KUKA KRL program: EPS_2_251292_SANCTRLMH1A_A_20251205052954.src

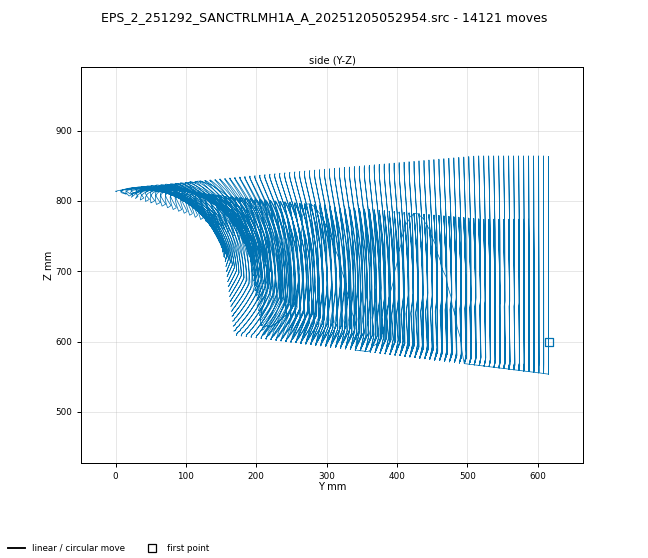
[picture p0: tool path of EPS_2_251292_SANCTRLMH1A_A_20251205052954.src, 14121 of 14123 moves have a stored position in this frame; points joined in program order, loops and branches not executed]
&ACCESS RVP
&REL 4
&COMMENT QRS 19112012
&PARAM EDITMASK = *
DEF PART()
EXT BAS (BAS_COMMAND :IN,REAL :IN )
INT I
BAS (#INITMOV,0 )

;KUKA QRS Post kuka4.cps  Date:22-06-2017 !

File_ID=2942

QRS_PRE_INIT()

;Init var - Until changes are made in qrs_pre_init
Outlet_Square_prg=0
Inlet_1_Square_prg=0
Inlet_2_Square_prg=0
Inlet_3_Square_prg=0
Inlet_4_Square_prg=0
Inlet_5_Square_prg=0

Outlet_1={X 0.000, Y 513.730, Z 763.500, B 0.000, E1 0.000 }
Inlet_1={X 0.000, Y 520.160, Z 673.500, B 0.000, E1 168.000 }
Inlet_2={X 0.000, Y 520.160, Z 673.500, B 0.000, E1 226.000 }
Outlet_1_type=201
Inlet_1_type=201
Inlet_2_type=201
;QRS#1=Sidecore dimensions
;QRS#2=200-8" PVC SDR 35
;QRS#3=200-8" PVC SDR 35
;QRS#4=200-8" PVC SDR 35
;QRS#5=
;QRS#6=
;QRS#7=
;QRS#8=
;QRS#9=12-08 PSX
;QRS#10=12-08 PSX
;QRS#11=12-08 PSX
;QRS#12=
;QRS#13=
;QRS#14=
;QRS#15=
;QRS#16=1220x127x1143 3,75'
;QRS#17=EPS Height
;QRS#18=864
;QRS#19=*
;QRS#20= UPDATED VERSION 22-06-2017
;QRS#21=*
Outlet_Square=0100
Inlet_1_Square=0100
Inlet_2_Square=0100
Inlet_3_Square=0
Inlet_4_Square=0
Inlet_5_Square=0
Mill_Square=1
Outlet_Square_Prg=204
Inlet_1_Square_prg=204
Inlet_2_Square_prg=204

QRS_INIT()

$ADVANCE=5

; T1
PTP {E1 173.592,E2 173.592}
PTP {X 0,Y 615.51,A -85,B 0,C 180,E1 173.592,E2 173.592,E3 0,E4 0,E5 0,E6 0}
QRS_SPEED_INIT()
LIN {X 0,Y 615.51,Z 600,A -85,B 0,C 180,E1 173.592,E2 173.592,E3 0,E4 0,E5 0,E6 0} C_VEL
LIN {X 0,Y 615.51,Z 563.866,A -85,B 0,C 180,E1 173.592,E2 173.592} C_VEL
LIN {X 0,Y 615.51,Z 555.694,A -85,B 0,C 180,E1 173.592,E2 173.592} C_VEL
LIN {X 0,Y 615.492,Z 553.694,A -85,B 0,C 180,E1 173.406,E2 173.406} C_VEL
LIN {X 0,Y 615.478,Z 553.692,A -85,B 0,C 180,E1 170.801,E2 170.801} C_VEL
LIN {X 0,Y 615.485,Z 553.682,A -85,B 0,C 180,E1 168.139,E2 168.139} C_VEL
LIN {X 0,Y 615.482,Z 553.692,A -85,B 0,C 180,E1 165.451,E2 165.451} C_VEL
LIN {X 0,Y 615.481,Z 553.693,A -85,B 0,C 180,E1 162.729,E2 162.729} C_VEL
LIN {X 0,Y 615.485,Z 553.682,A -85,B 0,C 180,E1 159.967,E2 159.967} C_VEL
LIN {X 0,Y 615.487,Z 553.696,A -85,B 0,C 180,E1 157.155,E2 157.155} C_VEL
LIN {X 0,Y 615.484,Z 553.684,A -85,B 0,C 180,E1 154.284,E2 154.284} C_VEL
LIN {X 0,Y 615.476,Z 553.687,A -85,B 0,C 180,E1 151.549,E2 151.549} C_VEL
LIN {X 0,Y 615.483,Z 553.703,A -85,B 0,C 180,E1 148.912,E2 148.912} C_VEL
LIN {X 0,Y 615.496,Z 553.68,A -85,B 0,C 180,E1 145.978,E2 145.978} C_VEL
LIN {X 0,Y 615.482,Z 553.694,A -85,B 0,C 180,E1 143.062,E2 143.062} C_VEL
LIN {X 0,Y 615.477,Z 553.689,A -85,B 0,C 180,E1 140.249,E2 140.249} C_VEL
LIN {X 0,Y 615.488,Z 553.681,A -85,B 0,C 180,E1 137.647,E2 137.647} C_VEL
LIN {X 0,Y 615.479,Z 553.696,A -85,B 0,C 180,E1 134.93,E2 134.93} C_VEL
LIN {X 0,Y 615.477,Z 553.687,A -85,B 0,C 180,E1 132.079,E2 132.079} C_VEL
LIN {X 0,Y 615.493,Z 553.68,A -85,B 0,C 180,E1 129.749,E2 129.749} C_VEL
LIN {X 0,Y 615.477,Z 553.693,A -85,B 0,C 180,E1 126.935,E2 126.935} C_VEL
LIN {X 0,Y 615.489,Z 553.697,A -85,B 0,C 180,E1 124.7,E2 124.7} C_VEL
LIN {X 0,Y 615.484,Z 553.696,A -85,B 0,C 180,E1 122.33,E2 122.33} C_VEL
LIN {X 0,Y 615.493,Z 553.68,A -85,B 0,C 180,E1 119.405,E2 119.405} C_VEL
LIN {X 0,Y 615.477,Z 553.849,A -85,B 0,C 180,E1 116.93,E2 116.93} C_VEL
LIN {X 0,Y 615.484,Z 564.333,A -85,B 0,C 180,E1 114.811,E2 114.811} C_VEL
LIN {X 0,Y 615.489,Z 670.429,A -85,B 0,C 180,E1 113.533,E2 113.533} C_VEL
LIN {X 0,Y 615.487,Z 683.41,A -85,B 0,C 180,E1 113.244,E2 113.244} C_VEL
LIN {X 0,Y 615.487,Z 695.565,A -85,B 0,C 180,E1 112.844,E2 112.844} C_VEL
LIN {X 0,Y 615.488,Z 707.887,A -85,B 0,C 180,E1 112.294,E2 112.294} C_VEL
LIN {X 0,Y 615.482,Z 719.67,A -85,B 0,C 180,E1 111.607,E2 111.607} C_VEL
LIN {X 0,Y 615.499,Z 730.452,A -85,B 0,C 180,E1 110.817,E2 110.817} C_VEL
LIN {X 0,Y 615.497,Z 739.119,A -85,B 0,C 180,E1 110.032,E2 110.032} C_VEL
LIN {X 0,Y 615.496,Z 748.438,A -85,B 0,C 180,E1 108.991,E2 108.991} C_VEL
LIN {X 0,Y 615.498,Z 755.797,A -85,B 0,C 180,E1 107.956,E2 107.956} C_VEL
LIN {X 0,Y 615.496,Z 761.581,A -85,B 0,C 180,E1 106.928,E2 106.928} C_VEL
LIN {X 0,Y 615.496,Z 766.062,A -85,B 0,C 180,E1 105.905,E2 105.905} C_VEL
LIN {X 0,Y 615.495,Z 768.406,A -85,B 0,C 180,E1 105.225,E2 105.225} C_VEL
LIN {X 0,Y 615.497,Z 770.293,A -85,B 0,C 180,E1 104.548,E2 104.548} C_VEL
LIN {X 0,Y 615.495,Z 771.682,A -85,B 0,C 180,E1 103.874,E2 103.874} C_VEL
LIN {X 0,Y 615.499,Z 772.654,A -85,B 0,C 180,E1 103.201,E2 103.201} C_VEL
LIN {X 0,Y 615.495,Z 773.23,A -85,B 0,C 180,E1 102.53,E2 102.53} C_VEL
LIN {X 0,Y 615.496,Z 773.372,A -85,B 0,C 180,E1 101.86,E2 101.86} C_VEL
LIN {X 0,Y 615.495,Z 772.439,A -85,B 0,C 180,E1 100.527,E2 100.527} C_VEL
LIN {X 0,Y 615.499,Z 771.379,A -85,B 0,C 180,E1 99.862,E2 99.862} C_VEL
LIN {X 0,Y 615.495,Z 769.863,A -85,B 0,C 180,E1 99.198,E2 99.198} C_VEL
LIN {X 0,Y 615.495,Z 766.811,A -85,B 0,C 180,E1 98.206,E2 98.206} C_VEL
LIN {X 0,Y 615.496,Z 762.717,A -85,B 0,C 180,E1 97.215,E2 97.215} C_VEL
LIN {X 0,Y 615.496,Z 756.461,A -85,B 0,C 180,E1 96.063,E2 96.063} C_VEL
LIN {X 0,Y 615.496,Z 749.669,A -85,B 0,C 180,E1 95.077,E2 95.077} C_VEL
LIN {X 0,Y 615.499,Z 741.216,A -85,B 0,C 180,E1 94.092,E2 94.092} C_VEL
LIN {X 0,Y 615.497,Z 732.559,A -85,B 0,C 180,E1 93.273,E2 93.273} C_VEL
LIN {X 0,Y 615.496,Z 721.959,A -85,B 0,C 180,E1 92.454,E2 92.454} C_VEL
LIN {X 0,Y 615.487,Z 711.331,A -85,B 0,C 180,E1 91.799,E2 91.799} C_VEL
LIN {X 0,Y 615.492,Z 699.51,A -85,B 0,C 180,E1 91.227,E2 91.227} C_VEL
LIN {X 0,Y 615.478,Z 687.237,A -85,B 0,C 180,E1 90.777,E2 90.777} C_VEL
LIN {X 0,Y 615.474,Z 674.443,A -85,B 0,C 180,E1 90.45,E2 90.45} C_VEL
LIN {X 0,Y 615.483,Z 659.053,A -85,B 0,C 180,E1 90.225,E2 90.225} C_VEL
LIN {X 0,Y 615.487,Z 563.524,A -85,B 0,C 180,E1 89.1,E2 89.1} C_VEL
LIN {X 0,Y 615.477,Z 553.688,A -85,B 0,C 180,E1 87.341,E2 87.341} C_VEL
LIN {X 0,Y 615.485,Z 553.683,A -85,B 0,C 180,E1 84.759,E2 84.759} C_VEL
LIN {X 0,Y 615.484,Z 553.697,A -85,B 0,C 180,E1 82.125,E2 82.125} C_VEL
LIN {X 0,Y 615.477,Z 553.69,A -85,B 0,C 180,E1 79.473,E2 79.473} C_VEL
LIN {X 0,Y 615.497,Z 553.68,A -85,B 0,C 180,E1 76.799,E2 76.799} C_VEL
LIN {X 0,Y 615.487,Z 553.698,A -85,B 0,C 180,E1 74.095,E2 74.095} C_VEL
LIN {X 0,Y 615.477,Z 553.688,A -85,B 0,C 180,E1 71.354,E2 71.354} C_VEL
LIN {X 0,Y 615.492,Z 553.684,A -85,B 0,C 180,E1 68.569,E2 68.569} C_VEL
LIN {X 0,Y 615.497,Z 553.692,A -85,B 0,C 180,E1 65.729,E2 65.729} C_VEL
LIN {X 0,Y 615.479,Z 553.684,A -85,B 0,C 180,E1 62.823,E2 62.823} C_VEL
LIN {X 0,Y 615.48,Z 553.696,A -85,B 0,C 180,E1 60.207,E2 60.207} C_VEL
LIN {X 0,Y 615.488,Z 553.688,A -85,B 0,C 180,E1 58.542,E2 58.542} C_VEL
LIN {X 0,Y 615.478,Z 563.8,A -85,B 0,C 180,E1 56.801,E2 56.801} C_VEL
LIN {X 0,Y 615.49,Z 670.43,A -85,B 0,C 180,E1 55.533,E2 55.533} C_VEL
LIN {X 0,Y 615.491,Z 683.455,A -85,B 0,C 180,E1 55.243,E2 55.243} C_VEL
LIN {X 0,Y 615.489,Z 695.76,A -85,B 0,C 180,E1 54.837,E2 54.837} C_VEL
LIN {X 0,Y 615.493,Z 707.167,A -85,B 0,C 180,E1 54.331,E2 54.331} C_VEL
LIN {X 0,Y 615.478,Z 719.02,A -85,B 0,C 180,E1 53.65,E2 53.65} C_VEL
LIN {X 0,Y 615.498,Z 729.264,A -85,B 0,C 180,E1 52.911,E2 52.911} C_VEL
LIN {X 0,Y 615.495,Z 737.595,A -85,B 0,C 180,E1 52.181,E2 52.181} C_VEL
LIN {X 0,Y 615.496,Z 745.845,A -85,B 0,C 180,E1 51.307,E2 51.307} C_VEL
LIN {X 0,Y 615.494,Z 753.849,A -85,B 0,C 180,E1 50.252,E2 50.252} C_VEL
LIN {X 0,Y 615.495,Z 760.453,A -85,B 0,C 180,E1 49.151,E2 49.151} C_VEL
LIN {X 0,Y 615.495,Z 764.795,A -85,B 0,C 180,E1 48.224,E2 48.224} C_VEL
LIN {X 0,Y 615.495,Z 768.162,A -85,B 0,C 180,E1 47.302,E2 47.302} C_VEL
LIN {X 0,Y 615.493,Z 771.468,A -85,B 0,C 180,E1 46.002,E2 46.002} C_VEL
LIN {X 0,Y 615.493,Z 772.946,A -85,B 0,C 180,E1 44.933,E2 44.933} C_VEL
LIN {X 0,Y 615.492,Z 773.385,A -85,B 0,C 180,E1 43.999,E2 43.999} C_VEL
LIN {X 0,Y 615.494,Z 772.997,A -85,B 0,C 180,E1 43.05,E2 43.05} C_VEL
LIN {X 0,Y 615.494,Z 771.759,A -85,B 0,C 180,E1 42.082,E2 42.082} C_VEL
LIN {X 0,Y 615.495,Z 769.591,A -85,B 0,C 180,E1 41.097,E2 41.097} C_VEL
LIN {X 0,Y 615.496,Z 766.384,A -85,B 0,C 180,E1 40.092,E2 40.092} C_VEL
LIN {X 0,Y 615.494,Z 761.199,A -85,B 0,C 180,E1 38.904,E2 38.904} C_VEL
LIN {X 0,Y 615.497,Z 754.943,A -85,B 0,C 180,E1 37.82,E2 37.82} C_VEL
LIN {X 0,Y 615.493,Z 747.546,A -85,B 0,C 180,E1 36.81,E2 36.81} C_VEL
LIN {X 0,Y 615.498,Z 738.717,A -85,B 0,C 180,E1 35.837,E2 35.837} C_VEL
LIN {X 0,Y 615.497,Z 729.459,A -85,B 0,C 180,E1 35.014,E2 35.014} C_VEL
LIN {X 0,Y 615.49,Z 719.279,A -85,B 0,C 180,E1 34.277,E2 34.277} C_VEL
LIN {X 0,Y 615.48,Z 707.513,A -85,B 0,C 180,E1 33.596,E2 33.596} C_VEL
LIN {X 0,Y 615.49,Z 696.199,A -85,B 0,C 180,E1 33.09,E2 33.09} C_VEL
LIN {X 0,Y 615.478,Z 684.677,A -85,B 0,C 180,E1 32.701,E2 32.701} C_VEL
LIN {X 0,Y 615.478,Z 671.437,A -85,B 0,C 180,E1 32.395,E2 32.395} C_VEL
LIN {X 0,Y 615.489,Z 640.455,A -85,B 0,C 180,E1 32.008,E2 32.008} C_VEL
LIN {X 0,Y 615.486,Z 564.37,A -85,B 0,C 180,E1 31.107,E2 31.107} C_VEL
LIN {X 0,Y 615.49,Z 553.686,A -85,B 0,C 180,E1 28.938,E2 28.938} C_VEL
LIN {X 0,Y 615.476,Z 553.684,A -85,B 0,C 180,E1 26.445,E2 26.445} C_VEL
LIN {X 0,Y 615.485,Z 553.686,A -85,B 0,C 180,E1 24.011,E2 24.011} C_VEL
LIN {X 0,Y 615.499,Z 553.699,A -85,B 0,C 180,E1 21.432,E2 21.432} C_VEL
LIN {X 0,Y 615.483,Z 553.683,A -85,B 0,C 180,E1 18.608,E2 18.608} C_VEL
LIN {X 0,Y 615.483,Z 553.689,A -85,B 0,C 180,E1 15.905,E2 15.905} C_VEL
LIN {X 0,Y 615.488,Z 553.693,A -85,B 0,C 180,E1 13.201,E2 13.201} C_VEL
LIN {X 0,Y 615.485,Z 553.682,A -85,B 0,C 180,E1 10.527,E2 10.527} C_VEL
LIN {X 0,Y 615.482,Z 553.69,A -85,B 0,C 180,E1 7.876,E2 7.876} C_VEL
LIN {X 0,Y 615.486,Z 553.695,A -85,B 0,C 180,E1 5.241,E2 5.241} C_VEL
LIN {X 0,Y 615.494,Z 553.681,A -85,B 0,C 180,E1 2.618,E2 2.618} C_VEL
LIN {X 0,Y 615.476,Z 553.689,A -85,B 0,C 180,E1 0,E2 0} C_VEL
LIN {X 0,Y 615.494,Z 553.698,A -85,B 0,C 180,E1 -2.618,E2 -2.618} C_VEL
LIN {X 0,Y 615.478,Z 553.686,A -85,B 0,C 180,E1 -5.241,E2 -5.241} C_VEL
LIN {X 0,Y 615.485,Z 553.685,A -85,B 0,C 180,E1 -7.876,E2 -7.876} C_VEL
LIN {X 0,Y 615.493,Z 553.701,A -85,B 0,C 180,E1 -10.527,E2 -10.527} C_VEL
LIN {X 0,Y 615.476,Z 553.687,A -85,B 0,C 180,E1 -13.202,E2 -13.202} C_VEL
LIN {X 0,Y 615.487,Z 553.685,A -85,B 0,C 180,E1 -15.905,E2 -15.905} C_VEL
LIN {X 0,Y 615.493,Z 553.696,A -85,B 0,C 180,E1 -18.646,E2 -18.646} C_VEL
LIN {X 0,Y 615.476,Z 553.684,A -85,B 0,C 180,E1 -21.432,E2 -21.432} C_VEL
LIN {X 0,Y 615.492,Z 553.693,A -85,B 0,C 180,E1 -24.272,E2 -24.272} C_VEL
LIN {X 0,Y 615.48,Z 553.686,A -85,B 0,C 180,E1 -27.178,E2 -27.178} C_VEL
LIN {X 0,Y 615.485,Z 553.684,A -85,B 0,C 180,E1 -29.797,E2 -29.797} C_VEL
LIN {X 0,Y 615.494,Z 553.7,A -85,B 0,C 180,E1 -32.457,E2 -32.457} C_VEL
LIN {X 0,Y 615.485,Z 553.692,A -85,B 0,C 180,E1 -34.815,E2 -34.815} C_VEL
LIN {X 0,Y 615.49,Z 553.683,A -85,B 0,C 180,E1 -37.242,E2 -37.242} C_VEL
LIN {X 0,Y 615.493,Z 553.688,A -85,B 0,C 180,E1 -40.091,E2 -40.091} C_VEL
LIN {X 0,Y 615.485,Z 553.687,A -85,B 0,C 180,E1 -43.049,E2 -43.049} C_VEL
LIN {X 0,Y 615.477,Z 553.687,A -85,B 0,C 180,E1 -45.851,E2 -45.851} C_VEL
LIN {X 0,Y 615.49,Z 553.701,A -85,B 0,C 180,E1 -48.528,E2 -48.528} C_VEL
LIN {X 0,Y 615.482,Z 553.686,A -85,B 0,C 180,E1 -51.096,E2 -51.096} C_VEL
LIN {X 0,Y 615.481,Z 553.683,A -85,B 0,C 180,E1 -53.576,E2 -53.576} C_VEL
LIN {X 0,Y 615.498,Z 553.7,A -85,B 0,C 180,E1 -56.465,E2 -56.465} C_VEL
LIN {X 0,Y 615.477,Z 553.688,A -85,B 0,C 180,E1 -59.081,E2 -59.081} C_VEL
LIN {X 0,Y 615.494,Z 553.68,A -85,B 0,C 180,E1 -61.549,E2 -61.549} C_VEL
LIN {X 0,Y 615.494,Z 553.7,A -85,B 0,C 180,E1 -64.43,E2 -64.43} C_VEL
LIN {X 0,Y 615.491,Z 553.765,A -85,B 0,C 180,E1 -65.706,E2 -65.706} C_VEL
LIN {X 0,Y 615.495,Z 577.471,A -85,B 0,C 180,E1 -68.569,E2 -68.569} C_VEL
LIN {X 0,Y 615.483,Z 601.351,A -85,B 0,C 180,E1 -71.397,E2 -71.397} C_VEL
LIN {X 0,Y 615.478,Z 624.467,A -85,B 0,C 180,E1 -74.095,E2 -74.095} C_VEL
LIN {X 0,Y 615.486,Z 649.386,A -85,B 0,C 180,E1 -76.967,E2 -76.967} C_VEL
LIN {X 0,Y 615.48,Z 650.668,A -85,B 0,C 180,E1 -77.114,E2 -77.114} C_VEL
LIN {X 0,Y 615.476,Z 759.849,A -85,B 0,C 180,E1 -78.411,E2 -78.411} C_VEL
LIN {X 0,Y 615.487,Z 772.354,A -85,B 0,C 180,E1 -78.682,E2 -78.682} C_VEL
LIN {X 0,Y 615.496,Z 785.511,A -85,B 0,C 180,E1 -79.109,E2 -79.109} C_VEL
LIN {X 0,Y 615.484,Z 797.482,A -85,B 0,C 180,E1 -79.64,E2 -79.64} C_VEL
LIN {X 0,Y 615.483,Z 809,A -85,B 0,C 180,E1 -80.304,E2 -80.304} C_VEL
LIN {X 0,Y 615.499,Z 819.344,A -85,B 0,C 180,E1 -81.05,E2 -81.05} C_VEL
LIN {X 0,Y 615.497,Z 827.814,A -85,B 0,C 180,E1 -81.794,E2 -81.794} C_VEL
LIN {X 0,Y 615.498,Z 835.608,A -85,B 0,C 180,E1 -82.62,E2 -82.62} C_VEL
LIN {X 0,Y 615.496,Z 843.204,A -85,B 0,C 180,E1 -83.608,E2 -83.608} C_VEL
LIN {X 0,Y 615.498,Z 850.205,A -85,B 0,C 180,E1 -84.759,E2 -84.759} C_VEL
LIN {X 0,Y 615.494,Z 854.852,A -85,B 0,C 180,E1 -85.744,E2 -85.744} C_VEL
LIN {X 0,Y 615.496,Z 858.399,A -85,B 0,C 180,E1 -86.727,E2 -86.727} C_VEL
LIN {X 0,Y 615.497,Z 860.233,A -85,B 0,C 180,E1 -87.382,E2 -87.382} C_VEL
LIN {X 0,Y 615.496,Z 861.608,A -85,B 0,C 180,E1 -88.037,E2 -88.037} C_VEL
LIN {X 0,Y 615.496,Z 863.174,A -85,B 0,C 180,E1 -89.346,E2 -89.346} C_VEL
LIN {X 0,Y 615.494,Z 863.389,A -85,B 0,C 180,E1 -90,E2 -90} C_VEL
LIN {X 0,Y 615.496,Z 862.58,A -85,B 0,C 180,E1 -91.309,E2 -91.309} C_VEL
LIN {X 0,Y 615.496,Z 861.608,A -85,B 0,C 180,E1 -91.963,E2 -91.963} C_VEL
LIN {X 0,Y 615.497,Z 860.233,A -85,B 0,C 180,E1 -92.618,E2 -92.618} C_VEL
LIN {X 0,Y 615.496,Z 857.35,A -85,B 0,C 180,E1 -93.601,E2 -93.601} C_VEL
LIN {X 0,Y 615.498,Z 853.442,A -85,B 0,C 180,E1 -94.584,E2 -94.584} C_VEL
LIN {X 0,Y 615.499,Z 848.406,A -85,B 0,C 180,E1 -95.57,E2 -95.57} C_VEL
LIN {X 0,Y 615.496,Z 841.869,A -85,B 0,C 180,E1 -96.583,E2 -96.583} C_VEL
LIN {X 0,Y 615.497,Z 834.135,A -85,B 0,C 180,E1 -97.545,E2 -97.545} C_VEL
LIN {X 0,Y 615.498,Z 826.047,A -85,B 0,C 180,E1 -98.371,E2 -98.371} C_VEL
LIN {X 0,Y 615.499,Z 816.17,A -85,B 0,C 180,E1 -99.198,E2 -99.198} C_VEL
LIN {X 0,Y 615.487,Z 804.986,A -85,B 0,C 180,E1 -99.945,E2 -99.945} C_VEL
LIN {X 0,Y 615.483,Z 794.029,A -85,B 0,C 180,E1 -100.527,E2 -100.527} C_VEL
LIN {X 0,Y 615.496,Z 781.435,A -85,B 0,C 180,E1 -101.042,E2 -101.042} C_VEL
LIN {X 0,Y 615.484,Z 769.078,A -85,B 0,C 180,E1 -101.401,E2 -101.401} C_VEL
LIN {X 0,Y 615.479,Z 755.489,A -85,B 0,C 180,E1 -101.652,E2 -101.652} C_VEL
LIN {X 0,Y 615.479,Z 649.625,A -85,B 0,C 180,E1 -102.907,E2 -102.907} C_VEL
LIN {X 0,Y 615.48,Z 623.138,A -85,B 0,C 180,E1 -105.565,E2 -105.565} C_VEL
LIN {X 0,Y 615.498,Z 596.408,A -85,B 0,C 180,E1 -108.279,E2 -108.279} C_VEL
LIN {X 0,Y 615.486,Z 567.537,A -85,B 0,C 180,E1 -111.256,E2 -111.256} C_VEL
LIN {X 0,Y 615.478,Z 553.684,A -85,B 0,C 180,E1 -112.72,E2 -112.72} C_VEL
LIN {X 0,Y 615.493,Z 553.69,A -85,B 0,C 180,E1 -115.569,E2 -115.569} C_VEL
LIN {X 0,Y 615.494,Z 553.684,A -85,B 0,C 180,E1 -118.451,E2 -118.451} C_VEL
LIN {X 0,Y 615.473,Z 553.685,A -85,B 0,C 180,E1 -121.083,E2 -121.083} C_VEL
LIN {X 0,Y 615.496,Z 553.686,A -85,B 0,C 180,E1 -123.535,E2 -123.535} C_VEL
LIN {X 0,Y 615.485,Z 553.69,A -85,B 0,C 180,E1 -126.424,E2 -126.424} C_VEL
LIN {X 0,Y 615.476,Z 553.684,A -85,B 0,C 180,E1 -129.06,E2 -129.06} C_VEL
LIN {X 0,Y 615.482,Z 553.686,A -85,B 0,C 180,E1 -131.473,E2 -131.473} C_VEL
LIN {X 0,Y 615.497,Z 553.7,A -85,B 0,C 180,E1 -134.147,E2 -134.147} C_VEL
LIN {X 0,Y 615.484,Z 553.683,A -85,B 0,C 180,E1 -136.951,E2 -136.951} C_VEL
LIN {X 0,Y 615.497,Z 553.69,A -85,B 0,C 180,E1 -139.908,E2 -139.908} C_VEL
LIN {X 0,Y 615.491,Z 553.685,A -85,B 0,C 180,E1 -142.758,E2 -142.758} C_VEL
LIN {X 0,Y 615.473,Z 553.684,A -85,B 0,C 180,E1 -145.299,E2 -145.299} C_VEL
LIN {X 0,Y 615.478,Z 553.686,A -85,B 0,C 180,E1 -147.668,E2 -147.668} C_VEL
LIN {X 0,Y 615.497,Z 553.696,A -85,B 0,C 180,E1 -150.201,E2 -150.201} C_VEL
LIN {X 0,Y 615.488,Z 553.685,A -85,B 0,C 180,E1 -152.952,E2 -152.952} C_VEL
LIN {X 0,Y 615.478,Z 553.686,A -85,B 0,C 180,E1 -155.727,E2 -155.727} C_VEL
LIN {X 0,Y 615.478,Z 553.7,A -85,B 0,C 180,E1 -158.568,E2 -158.568} C_VEL
LIN {X 0,Y 615.483,Z 553.682,A -85,B 0,C 180,E1 -161.392,E2 -161.392} C_VEL
LIN {X 0,Y 615.484,Z 553.689,A -85,B 0,C 180,E1 -164.095,E2 -164.095} C_VEL
LIN {X 0,Y 615.476,Z 553.696,A -85,B 0,C 180,E1 -166.798,E2 -166.798} C_VEL
LIN {X 0,Y 615.484,Z 553.682,A -85,B 0,C 180,E1 -169.473,E2 -169.473} C_VEL
LIN {X 0,Y 615.482,Z 553.688,A -85,B 0,C 180,E1 -172.124,E2 -172.124} C_VEL
LIN {X 0,Y 615.487,Z 553.699,A -85,B 0,C 180,E1 -174.759,E2 -174.759} C_VEL
LIN {X 0,Y 615.494,Z 553.682,A -85,B 0,C 180,E1 -177.382,E2 -177.382} C_VEL
LIN {X 0,Y 615.476,Z 553.686,A -85,B 0,C 180,E1 -180,E2 -180} C_VEL
LIN {X 0,Y 615.495,Z 553.696,A -85,B 0,C 180,E1 -182.618,E2 -182.618} C_VEL
LIN {X 0,Y 615.481,Z 553.689,A -85,B 0,C 180,E1 -185.241,E2 -185.241} C_VEL
LIN {X 0,Y 615.492,Z 553.694,A -85,B 0,C 180,E1 -186.594,E2 -186.594} C_VEL
LIN {X 0,Y 614.806,Z 553.839,A -85,B 0,C 180,E1 -187.14,E2 -187.14} C_VEL
LIN {X 0,Y 611.964,Z 554.25,A -85,B 0,C 180,E1 -188.026,E2 -188.026} C_VEL
LIN {X 0,Y 609.572,Z 554.562,A -85,B 0,C 180,E1 -188.738,E2 -188.738} C_VEL
LIN {X 0,Y 608.54,Z 554.68,A -85,B 0,C 180,E1 -189.288,E2 -189.288} C_VEL
LIN {X 0,Y 608.453,Z 554.688,A -85,B 0,C 180,E1 -189.474,E2 -189.474} C_VEL
LIN {X 0,Y 608.46,Z 554.686,A -85,B 0,C 180,E1 -192,E2 -192} C_VEL
LIN {X 0,Y 608.469,Z 554.692,A -85,B 0,C 180,E1 -194.721,E2 -194.721} C_VEL
LIN {X 0,Y 608.448,Z 554.69,A -85,B 0,C 180,E1 -197.477,E2 -197.477} C_VEL
LIN {X 0,Y 608.459,Z 554.687,A -85,B 0,C 180,E1 -200.274,E2 -200.274} C_VEL
LIN {X 0,Y 608.448,Z 554.697,A -85,B 0,C 180,E1 -203.124,E2 -203.124} C_VEL
LIN {X 0,Y 608.467,Z 554.686,A -85,B 0,C 180,E1 -205.723,E2 -205.723} C_VEL
LIN {X 0,Y 608.445,Z 554.688,A -85,B 0,C 180,E1 -208.267,E2 -208.267} C_VEL
LIN {X 0,Y 608.47,Z 554.687,A -85,B 0,C 180,E1 -210.545,E2 -210.545} C_VEL
LIN {X 0,Y 608.451,Z 554.693,A -85,B 0,C 180,E1 -212.88,E2 -212.88} C_VEL
LIN {X 0,Y 608.435,Z 554.698,A -85,B 0,C 180,E1 -215.278,E2 -215.278} C_VEL
LIN {X 0,Y 608.472,Z 554.687,A -85,B 0,C 180,E1 -217.746,E2 -217.746} C_VEL
LIN {X 0,Y 608.45,Z 554.687,A -85,B 0,C 180,E1 -220.33,E2 -220.33} C_VEL
LIN {X 0,Y 608.484,Z 554.694,A -85,B 0,C 180,E1 -223.312,E2 -223.312} C_VEL
LIN {X 0,Y 608.465,Z 554.685,A -85,B 0,C 180,E1 -226.132,E2 -226.132} C_VEL
LIN {X 0,Y 608.447,Z 554.69,A -85,B 0,C 180,E1 -228.824,E2 -228.824} C_VEL
LIN {X 0,Y 608.463,Z 554.696,A -85,B 0,C 180,E1 -231.413,E2 -231.413} C_VEL
LIN {X 0,Y 608.474,Z 554.687,A -85,B 0,C 180,E1 -233.951,E2 -233.951} C_VEL
LIN {X 0,Y 608.466,Z 554.685,A -85,B 0,C 180,E1 -236.33,E2 -236.33} C_VEL
LIN {X 0,Y 608.444,Z 554.689,A -85,B 0,C 180,E1 -238.733,E2 -238.733} C_VEL
LIN {X 0,Y 608.474,Z 554.693,A -85,B 0,C 180,E1 -241.38,E2 -241.38} C_VEL
LIN {X 0,Y 608.454,Z 554.736,A -85,B 0,C 180,E1 -243.037,E2 -243.037} C_VEL
LIN {X 0,Y 608.49,Z 564.85,A -85,B 0,C 180,E1 -245.061,E2 -245.061} C_VEL
LIN {X 0,Y 608.559,Z 669.713,A -85,B 0,C 180,E1 -246.318,E2 -246.318} C_VEL
LIN {X 0,Y 608.525,Z 682.964,A -85,B 0,C 180,E1 -246.61,E2 -246.61} C_VEL
LIN {X 0,Y 608.508,Z 695.282,A -85,B 0,C 180,E1 -247.014,E2 -247.014} C_VEL
LIN {X 0,Y 608.528,Z 706.51,A -85,B 0,C 180,E1 -247.509,E2 -247.509} C_VEL
LIN {X 0,Y 608.465,Z 717.598,A -85,B 0,C 180,E1 -248.131,E2 -248.131} C_VEL
LIN {X 0,Y 608.487,Z 728.844,A -85,B 0,C 180,E1 -248.932,E2 -248.932} C_VEL
LIN {X 0,Y 608.479,Z 737.934,A -85,B 0,C 180,E1 -249.727,E2 -249.727} C_VEL
LIN {X 0,Y 608.45,Z 746.187,A -85,B 0,C 180,E1 -250.605,E2 -250.605} C_VEL
LIN {X 0,Y 608.451,Z 754.193,A -85,B 0,C 180,E1 -251.664,E2 -251.664} C_VEL
LIN {X 0,Y 608.451,Z 759.485,A -85,B 0,C 180,E1 -252.524,E2 -252.524} C_VEL
LIN {X 0,Y 608.43,Z 764.279,A -85,B 0,C 180,E1 -253.484,E2 -253.484} C_VEL
LIN {X 0,Y 608.424,Z 768.507,A -85,B 0,C 180,E1 -254.593,E2 -254.593} C_VEL
LIN {X 0,Y 608.421,Z 770.495,A -85,B 0,C 180,E1 -255.279,E2 -255.279} C_VEL
LIN {X 0,Y 608.442,Z 772.093,A -85,B 0,C 180,E1 -255.994,E2 -255.994} C_VEL
LIN {X 0,Y 608.418,Z 773.741,A -85,B 0,C 180,E1 -257.322,E2 -257.322} C_VEL
LIN {X 0,Y 608.44,Z 773.995,A -85,B 0,C 180,E1 -258,E2 -258} C_VEL
LIN {X 0,Y 608.45,Z 773.538,A -85,B 0,C 180,E1 -259.055,E2 -259.055} C_VEL
LIN {X 0,Y 608.434,Z 772.215,A -85,B 0,C 180,E1 -260.023,E2 -260.023} C_VEL
LIN {X 0,Y 608.423,Z 770.808,A -85,B 0,C 180,E1 -260.694,E2 -260.694} C_VEL
LIN {X 0,Y 608.455,Z 767.858,A -85,B 0,C 180,E1 -261.699,E2 -261.699} C_VEL
LIN {X 0,Y 608.46,Z 763.872,A -85,B 0,C 180,E1 -262.701,E2 -262.701} C_VEL
LIN {X 0,Y 608.445,Z 757.966,A -85,B 0,C 180,E1 -263.831,E2 -263.831} C_VEL
LIN {X 0,Y 608.445,Z 751.089,A -85,B 0,C 180,E1 -264.864,E2 -264.864} C_VEL
LIN {X 0,Y 608.473,Z 742.853,A -85,B 0,C 180,E1 -265.86,E2 -265.86} C_VEL
LIN {X 0,Y 608.465,Z 734.439,A -85,B 0,C 180,E1 -266.689,E2 -266.689} C_VEL
LIN {X 0,Y 608.489,Z 724.099,A -85,B 0,C 180,E1 -267.518,E2 -267.518} C_VEL
LIN {X 0,Y 608.488,Z 712.524,A -85,B 0,C 180,E1 -268.263,E2 -268.263} C_VEL
LIN {X 0,Y 608.517,Z 700.956,A -85,B 0,C 180,E1 -268.842,E2 -268.842} C_VEL
LIN {X 0,Y 608.513,Z 687.799,A -85,B 0,C 180,E1 -269.338,E2 -269.338} C_VEL
LIN {X 0,Y 608.538,Z 675.243,A -85,B 0,C 180,E1 -269.669,E2 -269.669} C_VEL
LIN {X 0,Y 608.546,Z 660.396,A -85,B 0,C 180,E1 -269.897,E2 -269.897} C_VEL
LIN {X 0,Y 608.467,Z 563.709,A -85,B 0,C 180,E1 -271.055,E2 -271.055} C_VEL
LIN {X 0,Y 608.455,Z 554.689,A -85,B 0,C 180,E1 -272.689,E2 -272.689} C_VEL
LIN {X 0,Y 608.465,Z 554.686,A -85,B 0,C 180,E1 -275.302,E2 -275.302} C_VEL
LIN {X 0,Y 608.476,Z 554.694,A -85,B 0,C 180,E1 -277.967,E2 -277.967} C_VEL
LIN {X 0,Y 608.457,Z 554.688,A -85,B 0,C 180,E1 -280.65,E2 -280.65} C_VEL
LIN {X 0,Y 608.471,Z 554.686,A -85,B 0,C 180,E1 -283.356,E2 -283.356} C_VEL
LIN {X 0,Y 608.462,Z 554.696,A -85,B 0,C 180,E1 -286.093,E2 -286.093} C_VEL
LIN {X 0,Y 608.453,Z 554.687,A -85,B 0,C 180,E1 -288.869,E2 -288.869} C_VEL
LIN {X 0,Y 608.476,Z 554.689,A -85,B 0,C 180,E1 -291.691,E2 -291.691} C_VEL
LIN {X 0,Y 608.455,Z 554.689,A -85,B 0,C 180,E1 -294.57,E2 -294.57} C_VEL
LIN {X 0,Y 608.473,Z 554.685,A -85,B 0,C 180,E1 -297.206,E2 -297.206} C_VEL
LIN {X 0,Y 608.466,Z 554.696,A -85,B 0,C 180,E1 -299.971,E2 -299.971} C_VEL
LIN {X 0,Y 608.464,Z 554.834,A -85,B 0,C 180,E1 -301.461,E2 -301.461} C_VEL
LIN {X 0,Y 608.468,Z 563.992,A -85,B 0,C 180,E1 -303.05,E2 -303.05} C_VEL
LIN {X 0,Y 608.555,Z 670.151,A -85,B 0,C 180,E1 -304.325,E2 -304.325} C_VEL
LIN {X 0,Y 608.531,Z 683.162,A -85,B 0,C 180,E1 -304.615,E2 -304.615} C_VEL
LIN {X 0,Y 608.526,Z 696.402,A -85,B 0,C 180,E1 -305.056,E2 -305.056} C_VEL
LIN {X 0,Y 608.499,Z 707.879,A -85,B 0,C 180,E1 -305.577,E2 -305.577} C_VEL
LIN {X 0,Y 608.476,Z 718.518,A -85,B 0,C 180,E1 -306.192,E2 -306.192} C_VEL
LIN {X 0,Y 608.471,Z 728.607,A -85,B 0,C 180,E1 -306.913,E2 -306.913} C_VEL
LIN {X 0,Y 608.468,Z 738.128,A -85,B 0,C 180,E1 -307.745,E2 -307.745} C_VEL
LIN {X 0,Y 608.449,Z 746.044,A -85,B 0,C 180,E1 -308.588,E2 -308.588} C_VEL
LIN {X 0,Y 608.437,Z 754.135,A -85,B 0,C 180,E1 -309.656,E2 -309.656} C_VEL
LIN {X 0,Y 608.437,Z 760.653,A -85,B 0,C 180,E1 -310.738,E2 -310.738} C_VEL
LIN {X 0,Y 608.45,Z 765.083,A -85,B 0,C 180,E1 -311.672,E2 -311.672} C_VEL
LIN {X 0,Y 608.439,Z 767.648,A -85,B 0,C 180,E1 -312.332,E2 -312.332} C_VEL
LIN {X 0,Y 608.432,Z 770.566,A -85,B 0,C 180,E1 -313.305,E2 -313.305} C_VEL
LIN {X 0,Y 608.418,Z 772.535,A -85,B 0,C 180,E1 -314.26,E2 -314.26} C_VEL
LIN {X 0,Y 608.414,Z 773.655,A -85,B 0,C 180,E1 -315.2,E2 -315.2} C_VEL
LIN {X 0,Y 608.426,Z 773.987,A -85,B 0,C 180,E1 -316.126,E2 -316.126} C_VEL
LIN {X 0,Y 608.433,Z 773.55,A -85,B 0,C 180,E1 -317.038,E2 -317.038} C_VEL
LIN {X 0,Y 608.422,Z 772.361,A -85,B 0,C 180,E1 -317.935,E2 -317.935} C_VEL
LIN {X 0,Y 608.432,Z 770.469,A -85,B 0,C 180,E1 -318.821,E2 -318.821} C_VEL
LIN {X 0,Y 608.445,Z 767.867,A -85,B 0,C 180,E1 -319.696,E2 -319.696} C_VEL
LIN {X 0,Y 608.453,Z 763.862,A -85,B 0,C 180,E1 -320.703,E2 -320.703} C_VEL
LIN {X 0,Y 608.434,Z 758.387,A -85,B 0,C 180,E1 -321.762,E2 -321.762} C_VEL
LIN {X 0,Y 608.443,Z 751.246,A -85,B 0,C 180,E1 -322.843,E2 -322.843} C_VEL
LIN {X 0,Y 608.46,Z 744.251,A -85,B 0,C 180,E1 -323.704,E2 -323.704} C_VEL
LIN {X 0,Y 608.46,Z 735.185,A -85,B 0,C 180,E1 -324.622,E2 -324.622} C_VEL
LIN {X 0,Y 608.479,Z 725.449,A -85,B 0,C 180,E1 -325.42,E2 -325.42} C_VEL
LIN {X 0,Y 608.482,Z 713.656,A -85,B 0,C 180,E1 -326.196,E2 -326.196} C_VEL
LIN {X 0,Y 608.499,Z 702.435,A -85,B 0,C 180,E1 -326.777,E2 -326.777} C_VEL
LIN {X 0,Y 608.533,Z 691.089,A -85,B 0,C 180,E1 -327.23,E2 -327.23} C_VEL
LIN {X 0,Y 608.526,Z 678.163,A -85,B 0,C 180,E1 -327.602,E2 -327.602} C_VEL
LIN {X 0,Y 608.529,Z 664.475,A -85,B 0,C 180,E1 -327.848,E2 -327.848} C_VEL
LIN {X 0,Y 608.469,Z 564.643,A -85,B 0,C 180,E1 -329.036,E2 -329.036} C_VEL
LIN {X 0,Y 608.478,Z 554.686,A -85,B 0,C 180,E1 -331.098,E2 -331.098} C_VEL
LIN {X 0,Y 608.449,Z 554.689,A -85,B 0,C 180,E1 -333.226,E2 -333.226} C_VEL
LIN {X 0,Y 608.466,Z 554.69,A -85,B 0,C 180,E1 -336.155,E2 -336.155} C_VEL
LIN {X 0,Y 608.46,Z 554.689,A -85,B 0,C 180,E1 -339.019,E2 -339.019} C_VEL
LIN {X 0,Y 608.449,Z 554.688,A -85,B 0,C 180,E1 -341.828,E2 -341.828} C_VEL
LIN {X 0,Y 608.471,Z 554.695,A -85,B 0,C 180,E1 -344.594,E2 -344.594} C_VEL
LIN {X 0,Y 608.475,Z 554.685,A -85,B 0,C 180,E1 -347.323,E2 -347.323} C_VEL
LIN {X 0,Y 608.454,Z 554.69,A -85,B 0,C 180,E1 -350.023,E2 -350.023} C_VEL
LIN {X 0,Y 608.478,Z 554.692,A -85,B 0,C 180,E1 -352.701,E2 -352.701} C_VEL
LIN {X 0,Y 608.467,Z 554.685,A -85,B 0,C 180,E1 -355.362,E2 -355.362} C_VEL
LIN {X 0,Y 608.446,Z 554.69,A -85,B 0,C 180,E1 -358.014,E2 -358.014} C_VEL
LIN {X 0,Y 608.479,Z 554.692,A -85,B 0,C 180,E1 -360.662,E2 -360.662} C_VEL
LIN {X 0,Y 608.473,Z 554.685,A -85,B 0,C 180,E1 -363.311,E2 -363.311} C_VEL
LIN {X 0,Y 608.479,Z 554.686,A -85,B 0,C 180,E1 -365.967,E2 -365.967} C_VEL
LIN {X 0,Y 608.459,Z 554.695,A -85,B 0,C 180,E1 -368.636,E2 -368.636} C_VEL
LIN {X 0,Y 608.468,Z 554.685,A -85,B 0,C 180,E1 -371.324,E2 -371.324} C_VEL
LIN {X 0,Y 608.459,Z 554.689,A -85,B 0,C 180,E1 -374.038,E2 -374.038} C_VEL
LIN {X 0,Y 608.47,Z 554.691,A -85,B 0,C 180,E1 -376.784,E2 -376.784} C_VEL
LIN {X 0,Y 608.446,Z 554.688,A -85,B 0,C 180,E1 -379.571,E2 -379.571} C_VEL
LIN {X 0,Y 608.484,Z 554.694,A -85,B 0,C 180,E1 -382.485,E2 -382.485} C_VEL
LIN {X 0,Y 608.448,Z 554.688,A -85,B 0,C 180,E1 -385.301,E2 -385.301} C_VEL
LIN {X 0,Y 608.446,Z 554.688,A -85,B 0,C 180,E1 -387.518,E2 -387.518} C_VEL
LIN {X 0,Y 608.468,Z 554.688,A -85,B 0,C 180,E1 -389.974,E2 -389.974} C_VEL
LIN {X 0,Y 608.466,Z 554.696,A -85,B 0,C 180,E1 -392.525,E2 -392.525} C_VEL
LIN {X 0,Y 608.437,Z 554.69,A -85,B 0,C 180,E1 -395.278,E2 -395.278} C_VEL
LIN {X 0,Y 608.471,Z 554.685,A -85,B 0,C 180,E1 -397.746,E2 -397.746} C_VEL
LIN {X 0,Y 608.476,Z 554.692,A -85,B 0,C 180,E1 -400.333,E2 -400.333} C_VEL
LIN {X 0,Y 608.483,Z 554.684,A -85,B 0,C 180,E1 -403.312,E2 -403.312} C_VEL
LIN {X 0,Y 608.466,Z 554.69,A -85,B 0,C 180,E1 -406.132,E2 -406.132} C_VEL
LIN {X 0,Y 608.449,Z 554.693,A -85,B 0,C 180,E1 -408.824,E2 -408.824} C_VEL
LIN {X 0,Y 608.464,Z 554.686,A -85,B 0,C 180,E1 -411.413,E2 -411.413} C_VEL
LIN {X 0,Y 608.444,Z 554.691,A -85,B 0,C 180,E1 -413.955,E2 -413.955} C_VEL
LIN {X 0,Y 608.467,Z 554.694,A -85,B 0,C 180,E1 -416.33,E2 -416.33} C_VEL
LIN {X 0,Y 608.444,Z 554.695,A -85,B 0,C 180,E1 -418.733,E2 -418.733} C_VEL
LIN {X 0,Y 608.473,Z 554.685,A -85,B 0,C 180,E1 -421.38,E2 -421.38} C_VEL
LIN {X 0,Y 608.473,Z 554.692,A -85,B 0,C 180,E1 -424.279,E2 -424.279} C_VEL
LIN {X 0,Y 608.487,Z 554.707,A -85,B 0,C 180,E1 -425.525,E2 -425.525} C_VEL
LIN {X 0,Y 608.633,Z 570.633,A -85,B 0,C 180,E1 -427.485,E2 -427.485} C_VEL
LIN {X 0,Y 608.566,Z 595.112,A -85,B 0,C 180,E1 -430.434,E2 -430.434} C_VEL
LIN {X 0,Y 608.521,Z 617.164,A -85,B 0,C 180,E1 -433.045,E2 -433.045} C_VEL
LIN {X 0,Y 608.508,Z 640.687,A -85,B 0,C 180,E1 -435.793,E2 -435.793} C_VEL
LIN {X 0,Y 608.486,Z 650.794,A -85,B 0,C 180,E1 -436.963,E2 -436.963} C_VEL
LIN {X 0,Y 608.531,Z 759.963,A -85,B 0,C 180,E1 -438.277,E2 -438.277} C_VEL
LIN {X 0,Y 608.535,Z 773.226,A -85,B 0,C 180,E1 -438.572,E2 -438.572} C_VEL
LIN {X 0,Y 608.543,Z 786.341,A -85,B 0,C 180,E1 -439.009,E2 -439.009} C_VEL
LIN {X 0,Y 608.501,Z 797.64,A -85,B 0,C 180,E1 -439.519,E2 -439.519} C_VEL
LIN {X 0,Y 608.474,Z 809.201,A -85,B 0,C 180,E1 -440.191,E2 -440.191} C_VEL
LIN {X 0,Y 608.485,Z 819.596,A -85,B 0,C 180,E1 -440.946,E2 -440.946} C_VEL
LIN {X 0,Y 608.475,Z 828.114,A -85,B 0,C 180,E1 -441.699,E2 -441.699} C_VEL
LIN {X 0,Y 608.471,Z 835.962,A -85,B 0,C 180,E1 -442.534,E2 -442.534} C_VEL
LIN {X 0,Y 608.461,Z 843.287,A -85,B 0,C 180,E1 -443.485,E2 -443.485} C_VEL
LIN {X 0,Y 608.45,Z 848.867,A -85,B 0,C 180,E1 -444.366,E2 -444.366} C_VEL
LIN {X 0,Y 608.432,Z 853.951,A -85,B 0,C 180,E1 -445.362,E2 -445.362} C_VEL
LIN {X 0,Y 608.449,Z 857.896,A -85,B 0,C 180,E1 -446.358,E2 -446.358} C_VEL
LIN {X 0,Y 608.425,Z 860.809,A -85,B 0,C 180,E1 -447.352,E2 -447.352} C_VEL
LIN {X 0,Y 608.441,Z 862.201,A -85,B 0,C 180,E1 -448.014,E2 -448.014} C_VEL
LIN {X 0,Y 608.438,Z 863.783,A -85,B 0,C 180,E1 -449.338,E2 -449.338} C_VEL
LIN {X 0,Y 608.434,Z 864,A -85,B 0,C 180,E1 -450,E2 -450} C_VEL
LIN {X 0,Y 608.448,Z 863.184,A -85,B 0,C 180,E1 -451.324,E2 -451.324} C_VEL
LIN {X 0,Y 608.441,Z 862.201,A -85,B 0,C 180,E1 -451.986,E2 -451.986} C_VEL
LIN {X 0,Y 608.425,Z 860.809,A -85,B 0,C 180,E1 -452.648,E2 -452.648} C_VEL
LIN {X 0,Y 608.449,Z 857.896,A -85,B 0,C 180,E1 -453.642,E2 -453.642} C_VEL
LIN {X 0,Y 608.432,Z 853.951,A -85,B 0,C 180,E1 -454.638,E2 -454.638} C_VEL
LIN {X 0,Y 608.437,Z 847.877,A -85,B 0,C 180,E1 -455.801,E2 -455.801} C_VEL
LIN {X 0,Y 608.462,Z 841.236,A -85,B 0,C 180,E1 -456.799,E2 -456.799} C_VEL
LIN {X 0,Y 608.455,Z 832.991,A -85,B 0,C 180,E1 -457.8,E2 -457.8} C_VEL
LIN {X 0,Y 608.472,Z 824.539,A -85,B 0,C 180,E1 -458.636,E2 -458.636} C_VEL
LIN {X 0,Y 608.471,Z 814.094,A -85,B 0,C 180,E1 -459.473,E2 -459.473} C_VEL
LIN {X 0,Y 608.487,Z 803.76,A -85,B 0,C 180,E1 -460.145,E2 -460.145} C_VEL
LIN {X 0,Y 608.521,Z 792.25,A -85,B 0,C 180,E1 -460.741,E2 -460.741} C_VEL
LIN {X 0,Y 608.538,Z 779.887,A -85,B 0,C 180,E1 -461.225,E2 -461.225} C_VEL
LIN {X 0,Y 608.536,Z 766.452,A -85,B 0,C 180,E1 -461.597,E2 -461.597} C_VEL
LIN {X 0,Y 608.543,Z 754.107,A -85,B 0,C 180,E1 -461.808,E2 -461.808} C_VEL
LIN {X 0,Y 608.494,Z 649.727,A -85,B 0,C 180,E1 -463.058,E2 -463.058} C_VEL
LIN {X 0,Y 608.52,Z 621.487,A -85,B 0,C 180,E1 -465.92,E2 -465.92} C_VEL
LIN {X 0,Y 608.57,Z 595.252,A -85,B 0,C 180,E1 -468.614,E2 -468.614} C_VEL
LIN {X 0,Y 608.644,Z 567.537,A -85,B 0,C 180,E1 -471.507,E2 -471.507} C_VEL
LIN {X 0,Y 608.464,Z 554.687,A -85,B 0,C 180,E1 -472.875,E2 -472.875} C_VEL
LIN {X 0,Y 608.478,Z 554.692,A -85,B 0,C 180,E1 -475.722,E2 -475.722} C_VEL
LIN {X 0,Y 608.475,Z 554.685,A -85,B 0,C 180,E1 -478.62,E2 -478.62} C_VEL
LIN {X 0,Y 608.458,Z 554.688,A -85,B 0,C 180,E1 -481.316,E2 -481.316} C_VEL
LIN {X 0,Y 608.48,Z 554.69,A -85,B 0,C 180,E1 -483.736,E2 -483.736} C_VEL
LIN {X 0,Y 608.477,Z 554.694,A -85,B 0,C 180,E1 -486.089,E2 -486.089} C_VEL
LIN {X 0,Y 608.465,Z 554.688,A -85,B 0,C 180,E1 -488.587,E2 -488.587} C_VEL
LIN {X 0,Y 608.456,Z 554.687,A -85,B 0,C 180,E1 -491.341,E2 -491.341} C_VEL
LIN {X 0,Y 608.463,Z 554.694,A -85,B 0,C 180,E1 -494.264,E2 -494.264} C_VEL
LIN {X 0,Y 608.451,Z 554.687,A -85,B 0,C 180,E1 -497.04,E2 -497.04} C_VEL
LIN {X 0,Y 608.453,Z 554.69,A -85,B 0,C 180,E1 -499.697,E2 -499.697} C_VEL
LIN {X 0,Y 608.475,Z 554.695,A -85,B 0,C 180,E1 -502.254,E2 -502.254} C_VEL
LIN {X 0,Y 608.469,Z 554.685,A -85,B 0,C 180,E1 -505.09,E2 -505.09} C_VEL
LIN {X 0,Y 608.462,Z 554.69,A -85,B 0,C 180,E1 -507.905,E2 -507.905} C_VEL
LIN {X 0,Y 608.48,Z 554.693,A -85,B 0,C 180,E1 -510.221,E2 -510.221} C_VEL
LIN {X 0,Y 608.446,Z 554.688,A -85,B 0,C 180,E1 -513.226,E2 -513.226} C_VEL
LIN {X 0,Y 608.475,Z 554.686,A -85,B 0,C 180,E1 -515.845,E2 -515.845} C_VEL
LIN {X 0,Y 608.46,Z 554.694,A -85,B 0,C 180,E1 -518.308,E2 -518.308} C_VEL
LIN {X 0,Y 608.45,Z 554.688,A -85,B 0,C 180,E1 -521.13,E2 -521.13} C_VEL
LIN {X 0,Y 608.456,Z 554.688,A -85,B 0,C 180,E1 -523.906,E2 -523.906} C_VEL
LIN {X 0,Y 608.456,Z 554.696,A -85,B 0,C 180,E1 -526.643,E2 -526.643} C_VEL
LIN {X 0,Y 608.462,Z 554.686,A -85,B 0,C 180,E1 -529.35,E2 -529.35} C_VEL
LIN {X 0,Y 608.474,Z 554.686,A -85,B 0,C 180,E1 -532.033,E2 -532.033} C_VEL
LIN {X 0,Y 608.464,Z 554.696,A -85,B 0,C 180,E1 -534.698,E2 -534.698} C_VEL
LIN {X 0,Y 608.483,Z 554.684,A -85,B 0,C 180,E1 -537.352,E2 -537.352} C_VEL
LIN {X 0,Y 608.466,Z 554.686,A -85,B 0,C 180,E1 -540,E2 -540} C_VEL
LIN {X 0,Y 608.483,Z 554.692,A -85,B 0,C 180,E1 -542.648,E2 -542.648} C_VEL
LIN {X 0,Y 608.46,Z 554.688,A -85,B 0,C 180,E1 -545.302,E2 -545.302} C_VEL
LIN {X 0,Y 608.474,Z 554.684,A -85,B 0,C 180,E1 -547.967,E2 -547.967} C_VEL
LIN {X 0,Y 608.453,Z 554.688,A -85,B 0,C 180,E1 -549.474,E2 -549.474} C_VEL
LIN {X 0,Y 607.777,Z 554.773,A -85,B 0,C 180,E1 -550.027,E2 -550.027} C_VEL
LIN {X 0,Y 604.923,Z 555.136,A -85,B 0,C 180,E1 -550.924,E2 -550.924} C_VEL
LIN {X 0,Y 602.52,Z 555.43,A -85,B 0,C 180,E1 -551.645,E2 -551.645} C_VEL
LIN {X 0,Y 601.489,Z 555.555,A -85,B 0,C 180,E1 -552.202,E2 -552.202} C_VEL
LIN {X 0,Y 601.406,Z 555.567,A -85,B 0,C 180,E1 -552.39,E2 -552.39} C_VEL
LIN {X 0,Y 601.423,Z 555.574,A -85,B 0,C 180,E1 -554.897,E2 -554.897} C_VEL
LIN {X 0,Y 601.426,Z 555.572,A -85,B 0,C 180,E1 -556.986,E2 -556.986} C_VEL
LIN {X 0,Y 601.401,Z 555.565,A -85,B 0,C 180,E1 -559.81,E2 -559.81} C_VEL
LIN {X 0,Y 601.403,Z 555.57,A -85,B 0,C 180,E1 -562.683,E2 -562.683} C_VEL
LIN {X 0,Y 601.401,Z 555.573,A -85,B 0,C 180,E1 -564.879,E2 -564.879} C_VEL
LIN {X 0,Y 601.417,Z 555.564,A -85,B 0,C 180,E1 -567.868,E2 -567.868} C_VEL
LIN {X 0,Y 601.44,Z 555.56,A -85,B 0,C 180,E1 -570.163,E2 -570.163} C_VEL
LIN {X 0,Y 601.414,Z 555.568,A -85,B 0,C 180,E1 -572.716,E2 -572.716} C_VEL
LIN {X 0,Y 601.403,Z 555.575,A -85,B 0,C 180,E1 -575.115,E2 -575.115} C_VEL
LIN {X 0,Y 601.432,Z 555.568,A -85,B 0,C 180,E1 -577.419,E2 -577.419} C_VEL
LIN {X 0,Y 601.408,Z 555.565,A -85,B 0,C 180,E1 -579.995,E2 -579.995} C_VEL
LIN {X 0,Y 601.41,Z 555.565,A -85,B 0,C 180,E1 -582.671,E2 -582.671} C_VEL
LIN {X 0,Y 601.421,Z 555.57,A -85,B 0,C 180,E1 -585.483,E2 -585.483} C_VEL
LIN {X 0,Y 601.418,Z 555.563,A -85,B 0,C 180,E1 -588.408,E2 -588.408} C_VEL
LIN {X 0,Y 601.43,Z 555.565,A -85,B 0,C 180,E1 -590.876,E2 -590.876} C_VEL
LIN {X 0,Y 601.44,Z 555.566,A -85,B 0,C 180,E1 -593.735,E2 -593.735} C_VEL
LIN {X 0,Y 601.427,Z 555.563,A -85,B 0,C 180,E1 -596.687,E2 -596.687} C_VEL
LIN {X 0,Y 601.41,Z 555.568,A -85,B 0,C 180,E1 -599.058,E2 -599.058} C_VEL
LIN {X 0,Y 601.434,Z 555.57,A -85,B 0,C 180,E1 -601.374,E2 -601.374} C_VEL
LIN {X 0,Y 601.399,Z 555.676,A -85,B 0,C 180,E1 -603.051,E2 -603.051} C_VEL
LIN {X 0,Y 601.413,Z 564.606,A -85,B 0,C 180,E1 -604.892,E2 -604.892} C_VEL
LIN {X 0,Y 601.672,Z 570.905,A -85,B 0,C 180,E1 -604.984,E2 -604.984} C_VEL
LIN {X 0,Y 601.612,Z 670.11,A -85,B 0,C 180,E1 -606.187,E2 -606.187} C_VEL
LIN {X 0,Y 601.572,Z 683.627,A -85,B 0,C 180,E1 -606.494,E2 -606.494} C_VEL
LIN {X 0,Y 601.547,Z 696.067,A -85,B 0,C 180,E1 -606.914,E2 -606.914} C_VEL
LIN {X 0,Y 601.533,Z 707.953,A -85,B 0,C 180,E1 -607.458,E2 -607.458} C_VEL
LIN {X 0,Y 601.452,Z 719.395,A -85,B 0,C 180,E1 -608.133,E2 -608.133} C_VEL
LIN {X 0,Y 601.449,Z 729.716,A -85,B 0,C 180,E1 -608.894,E2 -608.894} C_VEL
LIN {X 0,Y 601.442,Z 738.236,A -85,B 0,C 180,E1 -609.658,E2 -609.658} C_VEL
LIN {X 0,Y 601.391,Z 746.422,A -85,B 0,C 180,E1 -610.546,E2 -610.546} C_VEL
LIN {X 0,Y 601.365,Z 754.317,A -85,B 0,C 180,E1 -611.607,E2 -611.607} C_VEL
LIN {X 0,Y 601.371,Z 760.585,A -85,B 0,C 180,E1 -612.662,E2 -612.662} C_VEL
LIN {X 0,Y 601.354,Z 765.469,A -85,B 0,C 180,E1 -613.711,E2 -613.711} C_VEL
LIN {X 0,Y 601.341,Z 769.144,A -85,B 0,C 180,E1 -614.755,E2 -614.755} C_VEL
LIN {X 0,Y 601.35,Z 772.034,A -85,B 0,C 180,E1 -615.937,E2 -615.937} C_VEL
LIN {X 0,Y 601.324,Z 773.641,A -85,B 0,C 180,E1 -617.17,E2 -617.17} C_VEL
LIN {X 0,Y 601.342,Z 773.962,A -85,B 0,C 180,E1 -617.856,E2 -617.856} C_VEL
LIN {X 0,Y 601.351,Z 773.567,A -85,B 0,C 180,E1 -619.026,E2 -619.026} C_VEL
LIN {X 0,Y 601.329,Z 772.449,A -85,B 0,C 180,E1 -619.903,E2 -619.903} C_VEL
LIN {X 0,Y 601.337,Z 771.126,A -85,B 0,C 180,E1 -620.583,E2 -620.583} C_VEL
LIN {X 0,Y 601.361,Z 768.31,A -85,B 0,C 180,E1 -621.6,E2 -621.6} C_VEL
LIN {X 0,Y 601.359,Z 764.474,A -85,B 0,C 180,E1 -622.614,E2 -622.614} C_VEL
LIN {X 0,Y 601.375,Z 758.653,A -85,B 0,C 180,E1 -623.784,E2 -623.784} C_VEL
LIN {X 0,Y 601.384,Z 752.125,A -85,B 0,C 180,E1 -624.804,E2 -624.804} C_VEL
LIN {X 0,Y 601.409,Z 744.097,A -85,B 0,C 180,E1 -625.812,E2 -625.812} C_VEL
LIN {X 0,Y 601.411,Z 735.953,A -85,B 0,C 180,E1 -626.65,E2 -626.65} C_VEL
LIN {X 0,Y 601.457,Z 726.022,A -85,B 0,C 180,E1 -627.489,E2 -627.489} C_VEL
LIN {X 0,Y 601.482,Z 714.871,A -85,B 0,C 180,E1 -628.242,E2 -628.242} C_VEL
LIN {X 0,Y 601.51,Z 703.994,A -85,B 0,C 180,E1 -628.828,E2 -628.828} C_VEL
LIN {X 0,Y 601.544,Z 691.981,A -85,B 0,C 180,E1 -629.331,E2 -629.331} C_VEL
LIN {X 0,Y 601.568,Z 679.492,A -85,B 0,C 180,E1 -629.707,E2 -629.707} C_VEL
LIN {X 0,Y 601.619,Z 666.424,A -85,B 0,C 180,E1 -629.958,E2 -629.958} C_VEL
LIN {X 0,Y 601.567,Z 564.767,A -85,B 0,C 180,E1 -631.182,E2 -631.182} C_VEL
LIN {X 0,Y 601.421,Z 563.688,A -85,B 0,C 180,E1 -631.214,E2 -631.214} C_VEL
LIN {X 0,Y 601.423,Z 555.565,A -85,B 0,C 180,E1 -632.679,E2 -632.679} C_VEL
LIN {X 0,Y 601.428,Z 555.563,A -85,B 0,C 180,E1 -635.364,E2 -635.364} C_VEL
LIN {X 0,Y 601.439,Z 555.572,A -85,B 0,C 180,E1 -638.061,E2 -638.061} C_VEL
LIN {X 0,Y 601.424,Z 555.563,A -85,B 0,C 180,E1 -641.01,E2 -641.01} C_VEL
LIN {X 0,Y 601.424,Z 555.565,A -85,B 0,C 180,E1 -643.515,E2 -643.515} C_VEL
LIN {X 0,Y 601.44,Z 555.567,A -85,B 0,C 180,E1 -646.286,E2 -646.286} C_VEL
LIN {X 0,Y 601.418,Z 555.563,A -85,B 0,C 180,E1 -649.098,E2 -649.098} C_VEL
LIN {X 0,Y 601.422,Z 555.572,A -85,B 0,C 180,E1 -651.958,E2 -651.958} C_VEL
LIN {X 0,Y 601.443,Z 555.567,A -85,B 0,C 180,E1 -654.293,E2 -654.293} C_VEL
LIN {X 0,Y 601.447,Z 555.56,A -85,B 0,C 180,E1 -657.111,E2 -657.111} C_VEL
LIN {X 0,Y 601.418,Z 555.565,A -85,B 0,C 180,E1 -659.392,E2 -659.392} C_VEL
LIN {X 0,Y 601.436,Z 555.677,A -85,B 0,C 180,E1 -661.439,E2 -661.439} C_VEL
LIN {X 0,Y 601.414,Z 563.751,A -85,B 0,C 180,E1 -662.887,E2 -662.887} C_VEL
LIN {X 0,Y 601.674,Z 574.728,A -85,B 0,C 180,E1 -663.03,E2 -663.03} C_VEL
LIN {X 0,Y 601.599,Z 670.522,A -85,B 0,C 180,E1 -664.195,E2 -664.195} C_VEL
LIN {X 0,Y 601.574,Z 684.306,A -85,B 0,C 180,E1 -664.513,E2 -664.513} C_VEL
LIN {X 0,Y 601.538,Z 696.293,A -85,B 0,C 180,E1 -664.923,E2 -664.923} C_VEL
LIN {X 0,Y 601.512,Z 708.499,A -85,B 0,C 180,E1 -665.488,E2 -665.488} C_VEL
LIN {X 0,Y 601.469,Z 719.009,A -85,B 0,C 180,E1 -666.108,E2 -666.108} C_VEL
LIN {X 0,Y 601.457,Z 729.682,A -85,B 0,C 180,E1 -666.891,E2 -666.891} C_VEL
LIN {X 0,Y 601.432,Z 739.018,A -85,B 0,C 180,E1 -667.735,E2 -667.735} C_VEL
LIN {X 0,Y 601.376,Z 748.23,A -85,B 0,C 180,E1 -668.771,E2 -668.771} C_VEL
LIN {X 0,Y 601.372,Z 755.18,A -85,B 0,C 180,E1 -669.737,E2 -669.737} C_VEL
LIN {X 0,Y 601.344,Z 761.709,A -85,B 0,C 180,E1 -670.879,E2 -670.879} C_VEL
LIN {X 0,Y 601.358,Z 767.232,A -85,B 0,C 180,E1 -672.174,E2 -672.174} C_VEL
LIN {X 0,Y 601.336,Z 770.16,A -85,B 0,C 180,E1 -673.118,E2 -673.118} C_VEL
LIN {X 0,Y 601.34,Z 771.308,A -85,B 0,C 180,E1 -673.593,E2 -673.593} C_VEL
LIN {X 0,Y 601.329,Z 772.972,A -85,B 0,C 180,E1 -674.526,E2 -674.526} C_VEL
LIN {X 0,Y 601.329,Z 773.848,A -85,B 0,C 180,E1 -675.473,E2 -675.473} C_VEL
LIN {X 0,Y 601.34,Z 773.916,A -85,B 0,C 180,E1 -676.435,E2 -676.435} C_VEL
LIN {X 0,Y 601.341,Z 773.147,A -85,B 0,C 180,E1 -677.415,E2 -677.415} C_VEL
LIN {X 0,Y 601.326,Z 771.481,A -85,B 0,C 180,E1 -678.416,E2 -678.416} C_VEL
LIN {X 0,Y 601.328,Z 768.826,A -85,B 0,C 180,E1 -679.435,E2 -679.435} C_VEL
LIN {X 0,Y 601.331,Z 765.053,A -85,B 0,C 180,E1 -680.475,E2 -680.475} C_VEL
LIN {X 0,Y 601.338,Z 759.982,A -85,B 0,C 180,E1 -681.539,E2 -681.539} C_VEL
LIN {X 0,Y 601.37,Z 753.373,A -85,B 0,C 180,E1 -682.624,E2 -682.624} C_VEL
LIN {X 0,Y 601.393,Z 745.931,A -85,B 0,C 180,E1 -683.603,E2 -683.603} C_VEL
LIN {X 0,Y 601.4,Z 736.555,A -85,B 0,C 180,E1 -684.593,E2 -684.593} C_VEL
LIN {X 0,Y 601.456,Z 727.461,A -85,B 0,C 180,E1 -685.376,E2 -685.376} C_VEL
LIN {X 0,Y 601.488,Z 716.89,A -85,B 0,C 180,E1 -686.12,E2 -686.12} C_VEL
LIN {X 0,Y 601.516,Z 705.137,A -85,B 0,C 180,E1 -686.773,E2 -686.773} C_VEL
LIN {X 0,Y 601.563,Z 692.614,A -85,B 0,C 180,E1 -687.307,E2 -687.307} C_VEL
LIN {X 0,Y 601.571,Z 679.619,A -85,B 0,C 180,E1 -687.703,E2 -687.703} C_VEL
LIN {X 0,Y 601.586,Z 666.061,A -85,B 0,C 180,E1 -687.964,E2 -687.964} C_VEL
LIN {X 0,Y 601.61,Z 565.993,A -85,B 0,C 180,E1 -689.166,E2 -689.166} C_VEL
LIN {X 0,Y 601.394,Z 564.587,A -85,B 0,C 180,E1 -689.203,E2 -689.203} C_VEL
LIN {X 0,Y 601.442,Z 555.563,A -85,B 0,C 180,E1 -691.107,E2 -691.107} C_VEL
LIN {X 0,Y 601.399,Z 555.566,A -85,B 0,C 180,E1 -693.636,E2 -693.636} C_VEL
LIN {X 0,Y 601.42,Z 555.574,A -85,B 0,C 180,E1 -696.59,E2 -696.59} C_VEL
LIN {X 0,Y 601.426,Z 555.563,A -85,B 0,C 180,E1 -699.478,E2 -699.478} C_VEL
LIN {X 0,Y 601.399,Z 555.573,A -85,B 0,C 180,E1 -702.312,E2 -702.312} C_VEL
LIN {X 0,Y 601.426,Z 555.565,A -85,B 0,C 180,E1 -705.103,E2 -705.103} C_VEL
LIN {X 0,Y 601.416,Z 555.565,A -85,B 0,C 180,E1 -707.857,E2 -707.857} C_VEL
LIN {X 0,Y 601.414,Z 555.574,A -85,B 0,C 180,E1 -710.584,E2 -710.584} C_VEL
LIN {X 0,Y 601.444,Z 555.561,A -85,B 0,C 180,E1 -713.323,E2 -713.323} C_VEL
LIN {X 0,Y 601.4,Z 555.568,A -85,B 0,C 180,E1 -715.979,E2 -715.979} C_VEL
LIN {X 0,Y 601.424,Z 555.571,A -85,B 0,C 180,E1 -718.661,E2 -718.661} C_VEL
LIN {X 0,Y 601.421,Z 555.563,A -85,B 0,C 180,E1 -721.339,E2 -721.339} C_VEL
LIN {X 0,Y 601.404,Z 555.568,A -85,B 0,C 180,E1 -724.021,E2 -724.021} C_VEL
LIN {X 0,Y 601.441,Z 555.568,A -85,B 0,C 180,E1 -726.711,E2 -726.711} C_VEL
LIN {X 0,Y 601.41,Z 555.564,A -85,B 0,C 180,E1 -729.416,E2 -729.416} C_VEL
LIN {X 0,Y 601.419,Z 555.568,A -85,B 0,C 180,E1 -732.142,E2 -732.142} C_VEL
LIN {X 0,Y 601.428,Z 555.566,A -85,B 0,C 180,E1 -734.897,E2 -734.897} C_VEL
LIN {X 0,Y 601.425,Z 555.565,A -85,B 0,C 180,E1 -736.986,E2 -736.986} C_VEL
LIN {X 0,Y 601.404,Z 555.566,A -85,B 0,C 180,E1 -739.81,E2 -739.81} C_VEL
LIN {X 0,Y 601.447,Z 555.567,A -85,B 0,C 180,E1 -742.682,E2 -742.682} C_VEL
LIN {X 0,Y 601.402,Z 555.57,A -85,B 0,C 180,E1 -744.879,E2 -744.879} C_VEL
LIN {X 0,Y 601.421,Z 555.564,A -85,B 0,C 180,E1 -747.867,E2 -747.867} C_VEL
LIN {X 0,Y 601.441,Z 555.565,A -85,B 0,C 180,E1 -750.163,E2 -750.163} C_VEL
LIN {X 0,Y 601.424,Z 555.57,A -85,B 0,C 180,E1 -752.718,E2 -752.718} C_VEL
LIN {X 0,Y 601.406,Z 555.567,A -85,B 0,C 180,E1 -755.115,E2 -755.115} C_VEL
LIN {X 0,Y 601.431,Z 555.562,A -85,B 0,C 180,E1 -757.419,E2 -757.419} C_VEL
LIN {X 0,Y 601.412,Z 555.567,A -85,B 0,C 180,E1 -759.995,E2 -759.995} C_VEL
LIN {X 0,Y 601.434,Z 555.569,A -85,B 0,C 180,E1 -762.669,E2 -762.669} C_VEL
LIN {X 0,Y 601.421,Z 555.563,A -85,B 0,C 180,E1 -765.483,E2 -765.483} C_VEL
LIN {X 0,Y 601.421,Z 555.573,A -85,B 0,C 180,E1 -768.408,E2 -768.408} C_VEL
LIN {X 0,Y 601.431,Z 555.566,A -85,B 0,C 180,E1 -770.876,E2 -770.876} C_VEL
LIN {X 0,Y 601.398,Z 555.566,A -85,B 0,C 180,E1 -773.418,E2 -773.418} C_VEL
LIN {X 0,Y 601.433,Z 555.565,A -85,B 0,C 180,E1 -776.065,E2 -776.065} C_VEL
LIN {X 0,Y 601.419,Z 555.574,A -85,B 0,C 180,E1 -778.546,E2 -778.546} C_VEL
LIN {X 0,Y 601.433,Z 555.562,A -85,B 0,C 180,E1 -781.374,E2 -781.374} C_VEL
LIN {X 0,Y 601.414,Z 555.57,A -85,B 0,C 180,E1 -784.133,E2 -784.133} C_VEL
LIN {X 0,Y 601.437,Z 555.632,A -85,B 0,C 180,E1 -785.335,E2 -785.335} C_VEL
LIN {X 0,Y 601.823,Z 557.832,A -85,B 0,C 180,E1 -785.627,E2 -785.627} C_VEL
LIN {X 0,Y 601.703,Z 580.411,A -85,B 0,C 180,E1 -788.413,E2 -788.413} C_VEL
LIN {X 0,Y 601.61,Z 603.842,A -85,B 0,C 180,E1 -791.251,E2 -791.251} C_VEL
LIN {X 0,Y 601.539,Z 627.455,A -85,B 0,C 180,E1 -794.065,E2 -794.065} C_VEL
LIN {X 0,Y 601.481,Z 650.794,A -85,B 0,C 180,E1 -796.808,E2 -796.808} C_VEL
LIN {X 0,Y 601.616,Z 727.293,A -85,B 0,C 180,E1 -797.734,E2 -797.734} C_VEL
LIN {X 0,Y 601.614,Z 761.104,A -85,B 0,C 180,E1 -798.161,E2 -798.161} C_VEL
LIN {X 0,Y 601.569,Z 773.985,A -85,B 0,C 180,E1 -798.459,E2 -798.459} C_VEL
LIN {X 0,Y 601.574,Z 786.594,A -85,B 0,C 180,E1 -798.89,E2 -798.89} C_VEL
LIN {X 0,Y 601.524,Z 797.639,A -85,B 0,C 180,E1 -799.396,E2 -799.396} C_VEL
LIN {X 0,Y 601.477,Z 809.202,A -85,B 0,C 180,E1 -800.076,E2 -800.076} C_VEL
LIN {X 0,Y 601.444,Z 819.597,A -85,B 0,C 180,E1 -800.839,E2 -800.839} C_VEL
LIN {X 0,Y 601.429,Z 828.114,A -85,B 0,C 180,E1 -801.601,E2 -801.601} C_VEL
LIN {X 0,Y 601.418,Z 835.962,A -85,B 0,C 180,E1 -802.446,E2 -802.446} C_VEL
LIN {X 0,Y 601.37,Z 843.226,A -85,B 0,C 180,E1 -803.398,E2 -803.398} C_VEL
LIN {X 0,Y 601.371,Z 848.867,A -85,B 0,C 180,E1 -804.299,E2 -804.299} C_VEL
LIN {X 0,Y 601.336,Z 853.95,A -85,B 0,C 180,E1 -805.307,E2 -805.307} C_VEL
LIN {X 0,Y 601.368,Z 857.896,A -85,B 0,C 180,E1 -806.315,E2 -806.315} C_VEL
LIN {X 0,Y 601.325,Z 860.809,A -85,B 0,C 180,E1 -807.321,E2 -807.321} C_VEL
LIN {X 0,Y 601.34,Z 862.202,A -85,B 0,C 180,E1 -807.991,E2 -807.991} C_VEL
LIN {X 0,Y 601.339,Z 863.784,A -85,B 0,C 180,E1 -809.33,E2 -809.33} C_VEL
LIN {X 0,Y 601.335,Z 864,A -85,B 0,C 180,E1 -810,E2 -810} C_VEL
LIN {X 0,Y 601.348,Z 863.184,A -85,B 0,C 180,E1 -811.339,E2 -811.339} C_VEL
LIN {X 0,Y 601.34,Z 862.202,A -85,B 0,C 180,E1 -812.009,E2 -812.009} C_VEL
LIN {X 0,Y 601.325,Z 860.809,A -85,B 0,C 180,E1 -812.679,E2 -812.679} C_VEL
LIN {X 0,Y 601.368,Z 857.896,A -85,B 0,C 180,E1 -813.685,E2 -813.685} C_VEL
LIN {X 0,Y 601.336,Z 853.951,A -85,B 0,C 180,E1 -814.693,E2 -814.693} C_VEL
LIN {X 0,Y 601.372,Z 847.878,A -85,B 0,C 180,E1 -815.869,E2 -815.869} C_VEL
LIN {X 0,Y 601.382,Z 841.237,A -85,B 0,C 180,E1 -816.88,E2 -816.88} C_VEL
LIN {X 0,Y 601.4,Z 832.991,A -85,B 0,C 180,E1 -817.892,E2 -817.892} C_VEL
LIN {X 0,Y 601.436,Z 824.539,A -85,B 0,C 180,E1 -818.737,E2 -818.737} C_VEL
LIN {X 0,Y 601.44,Z 814.095,A -85,B 0,C 180,E1 -819.585,E2 -819.585} C_VEL
LIN {X 0,Y 601.489,Z 803.761,A -85,B 0,C 180,E1 -820.264,E2 -820.264} C_VEL
LIN {X 0,Y 601.536,Z 792.905,A -85,B 0,C 180,E1 -820.836,E2 -820.836} C_VEL
LIN {X 0,Y 601.567,Z 780.385,A -85,B 0,C 180,E1 -821.34,E2 -821.34} C_VEL
LIN {X 0,Y 601.596,Z 767.366,A -85,B 0,C 180,E1 -821.711,E2 -821.711} C_VEL
LIN {X 0,Y 601.61,Z 754.107,A -85,B 0,C 180,E1 -821.946,E2 -821.946} C_VEL
LIN {X 0,Y 601.562,Z 650.381,A -85,B 0,C 180,E1 -823.19,E2 -823.19} C_VEL
LIN {X 0,Y 601.485,Z 649.305,A -85,B 0,C 180,E1 -823.256,E2 -823.256} C_VEL
LIN {X 0,Y 601.577,Z 621.487,A -85,B 0,C 180,E1 -826.108,E2 -826.108} C_VEL
LIN {X 0,Y 601.649,Z 596.04,A -85,B 0,C 180,E1 -828.754,E2 -828.754} C_VEL
LIN {X 0,Y 601.771,Z 570.909,A -85,B 0,C 180,E1 -831.405,E2 -831.405} C_VEL
LIN {X 0,Y 601.832,Z 557.592,A -85,B 0,C 180,E1 -832.829,E2 -832.829} C_VEL
LIN {X 0,Y 601.418,Z 555.568,A -85,B 0,C 180,E1 -833.091,E2 -833.091} C_VEL
LIN {X 0,Y 601.438,Z 555.568,A -85,B 0,C 180,E1 -835.617,E2 -835.617} C_VEL
LIN {X 0,Y 601.422,Z 555.574,A -85,B 0,C 180,E1 -837.867,E2 -837.867} C_VEL
LIN {X 0,Y 601.428,Z 555.569,A -85,B 0,C 180,E1 -840.163,E2 -840.163} C_VEL
LIN {X 0,Y 601.422,Z 555.563,A -85,B 0,C 180,E1 -842.715,E2 -842.715} C_VEL
LIN {X 0,Y 601.412,Z 555.564,A -85,B 0,C 180,E1 -845.114,E2 -845.114} C_VEL
LIN {X 0,Y 601.431,Z 555.563,A -85,B 0,C 180,E1 -847.418,E2 -847.418} C_VEL
LIN {X 0,Y 601.413,Z 555.574,A -85,B 0,C 180,E1 -849.994,E2 -849.994} C_VEL
LIN {X 0,Y 601.406,Z 555.567,A -85,B 0,C 180,E1 -852.669,E2 -852.669} C_VEL
LIN {X 0,Y 601.421,Z 555.564,A -85,B 0,C 180,E1 -855.481,E2 -855.481} C_VEL
LIN {X 0,Y 601.425,Z 555.569,A -85,B 0,C 180,E1 -858.405,E2 -858.405} C_VEL
LIN {X 0,Y 601.436,Z 555.562,A -85,B 0,C 180,E1 -860.875,E2 -860.875} C_VEL
LIN {X 0,Y 601.439,Z 555.563,A -85,B 0,C 180,E1 -863.733,E2 -863.733} C_VEL
LIN {X 0,Y 601.422,Z 555.567,A -85,B 0,C 180,E1 -866.686,E2 -866.686} C_VEL
LIN {X 0,Y 601.426,Z 555.563,A -85,B 0,C 180,E1 -869.058,E2 -869.058} C_VEL
LIN {X 0,Y 601.424,Z 555.562,A -85,B 0,C 180,E1 -871.373,E2 -871.373} C_VEL
LIN {X 0,Y 601.416,Z 555.57,A -85,B 0,C 180,E1 -874.129,E2 -874.129} C_VEL
LIN {X 0,Y 601.418,Z 555.57,A -85,B 0,C 180,E1 -876.59,E2 -876.59} C_VEL
LIN {X 0,Y 601.426,Z 555.562,A -85,B 0,C 180,E1 -879.478,E2 -879.478} C_VEL
LIN {X 0,Y 601.393,Z 555.574,A -85,B 0,C 180,E1 -882.311,E2 -882.311} C_VEL
LIN {X 0,Y 601.409,Z 555.573,A -85,B 0,C 180,E1 -884.409,E2 -884.409} C_VEL
LIN {X 0,Y 601.416,Z 555.565,A -85,B 0,C 180,E1 -887.172,E2 -887.172} C_VEL
LIN {X 0,Y 601.431,Z 555.562,A -85,B 0,C 180,E1 -889.905,E2 -889.905} C_VEL
LIN {X 0,Y 601.446,Z 555.57,A -85,B 0,C 180,E1 -892.615,E2 -892.615} C_VEL
LIN {X 0,Y 601.433,Z 555.563,A -85,B 0,C 180,E1 -895.308,E2 -895.308} C_VEL
LIN {X 0,Y 601.417,Z 555.564,A -85,B 0,C 180,E1 -897.991,E2 -897.991} C_VEL
LIN {X 0,Y 601.455,Z 555.568,A -85,B 0,C 180,E1 -900.67,E2 -900.67} C_VEL
LIN {X 0,Y 601.425,Z 555.564,A -85,B 0,C 180,E1 -903.35,E2 -903.35} C_VEL
LIN {X 0,Y 601.426,Z 555.562,A -85,B 0,C 180,E1 -906.037,E2 -906.037} C_VEL
LIN {X 0,Y 601.435,Z 555.57,A -85,B 0,C 180,E1 -908.738,E2 -908.738} C_VEL
LIN {X 0,Y 601.427,Z 555.563,A -85,B 0,C 180,E1 -911.458,E2 -911.458} C_VEL
LIN {X 0,Y 601.406,Z 555.567,A -85,B 0,C 180,E1 -912.39,E2 -912.39} C_VEL
LIN {X 0,Y 600.741,Z 555.657,A -85,B 0,C 180,E1 -912.95,E2 -912.95} C_VEL
LIN {X 0,Y 597.888,Z 556.016,A -85,B 0,C 180,E1 -913.857,E2 -913.857} C_VEL
LIN {X 0,Y 595.476,Z 556.314,A -85,B 0,C 180,E1 -914.588,E2 -914.588} C_VEL
LIN {X 0,Y 594.439,Z 556.44,A -85,B 0,C 180,E1 -915.151,E2 -915.151} C_VEL
LIN {X 0,Y 594.354,Z 556.447,A -85,B 0,C 180,E1 -915.342,E2 -915.342} C_VEL
LIN {X 0,Y 594.374,Z 556.44,A -85,B 0,C 180,E1 -917.904,E2 -917.904} C_VEL
LIN {X 0,Y 594.374,Z 556.45,A -85,B 0,C 180,E1 -920.919,E2 -920.919} C_VEL
LIN {X 0,Y 594.386,Z 556.44,A -85,B 0,C 180,E1 -923.704,E2 -923.704} C_VEL
LIN {X 0,Y 594.384,Z 556.444,A -85,B 0,C 180,E1 -926.7,E2 -926.7} C_VEL
LIN {X 0,Y 594.374,Z 556.45,A -85,B 0,C 180,E1 -928.999,E2 -928.999} C_VEL
LIN {X 0,Y 594.385,Z 556.442,A -85,B 0,C 180,E1 -931.646,E2 -931.646} C_VEL
LIN {X 0,Y 594.386,Z 556.441,A -85,B 0,C 180,E1 -934.58,E2 -934.58} C_VEL
LIN {X 0,Y 594.382,Z 556.449,A -85,B 0,C 180,E1 -937.087,E2 -937.087} C_VEL
LIN {X 0,Y 594.371,Z 556.443,A -85,B 0,C 180,E1 -939.776,E2 -939.776} C_VEL
LIN {X 0,Y 594.367,Z 556.44,A -85,B 0,C 180,E1 -942.376,E2 -942.376} C_VEL
LIN {X 0,Y 594.359,Z 556.452,A -85,B 0,C 180,E1 -945.192,E2 -945.192} C_VEL
LIN {X 0,Y 594.377,Z 556.44,A -85,B 0,C 180,E1 -948.153,E2 -948.153} C_VEL
LIN {X 0,Y 594.382,Z 556.447,A -85,B 0,C 180,E1 -951.196,E2 -951.196} C_VEL
LIN {X 0,Y 594.392,Z 556.443,A -85,B 0,C 180,E1 -953.759,E2 -953.759} C_VEL
LIN {X 0,Y 594.379,Z 556.441,A -85,B 0,C 180,E1 -956.24,E2 -956.24} C_VEL
LIN {X 0,Y 594.368,Z 556.442,A -85,B 0,C 180,E1 -958.651,E2 -958.651} C_VEL
LIN {X 0,Y 594.384,Z 556.443,A -85,B 0,C 180,E1 -961.043,E2 -961.043} C_VEL
LIN {X 0,Y 594.354,Z 556.597,A -85,B 0,C 180,E1 -963.062,E2 -963.062} C_VEL
LIN {X 0,Y 594.354,Z 564.624,A -85,B 0,C 180,E1 -964.736,E2 -964.736} C_VEL
LIN {X 0,Y 594.763,Z 568.612,A -85,B 0,C 180,E1 -964.802,E2 -964.802} C_VEL
LIN {X 0,Y 594.666,Z 670.5,A -85,B 0,C 180,E1 -966.054,E2 -966.054} C_VEL
LIN {X 0,Y 594.621,Z 684.289,A -85,B 0,C 180,E1 -966.376,E2 -966.376} C_VEL
LIN {X 0,Y 594.571,Z 696.804,A -85,B 0,C 180,E1 -966.812,E2 -966.812} C_VEL
LIN {X 0,Y 594.506,Z 709.215,A -85,B 0,C 180,E1 -967.401,E2 -967.401} C_VEL
LIN {X 0,Y 594.45,Z 721.189,A -85,B 0,C 180,E1 -968.136,E2 -968.136} C_VEL
LIN {X 0,Y 594.404,Z 730.29,A -85,B 0,C 180,E1 -968.831,E2 -968.831} C_VEL
LIN {X 0,Y 594.35,Z 740.261,A -85,B 0,C 180,E1 -969.766,E2 -969.766} C_VEL
LIN {X 0,Y 594.34,Z 748.084,A -85,B 0,C 180,E1 -970.665,E2 -970.665} C_VEL
LIN {X 0,Y 594.316,Z 755.672,A -85,B 0,C 180,E1 -971.738,E2 -971.738} C_VEL
LIN {X 0,Y 594.278,Z 761.644,A -85,B 0,C 180,E1 -972.804,E2 -972.804} C_VEL
LIN {X 0,Y 594.256,Z 766.272,A -85,B 0,C 180,E1 -973.864,E2 -973.864} C_VEL
LIN {X 0,Y 594.244,Z 769.731,A -85,B 0,C 180,E1 -974.919,E2 -974.919} C_VEL
LIN {X 0,Y 594.261,Z 771.967,A -85,B 0,C 180,E1 -975.876,E2 -975.876} C_VEL
LIN {X 0,Y 594.243,Z 773.54,A -85,B 0,C 180,E1 -977.015,E2 -977.015} C_VEL
LIN {X 0,Y 594.239,Z 773.929,A -85,B 0,C 180,E1 -977.709,E2 -977.709} C_VEL
LIN {X 0,Y 594.25,Z 773.526,A -85,B 0,C 180,E1 -979.093,E2 -979.093} C_VEL
LIN {X 0,Y 594.232,Z 772.682,A -85,B 0,C 180,E1 -979.782,E2 -979.782} C_VEL
LIN {X 0,Y 594.256,Z 771.429,A -85,B 0,C 180,E1 -980.47,E2 -980.47} C_VEL
LIN {X 0,Y 594.26,Z 768.758,A -85,B 0,C 180,E1 -981.499,E2 -981.499} C_VEL
LIN {X 0,Y 594.277,Z 765.073,A -85,B 0,C 180,E1 -982.526,E2 -982.526} C_VEL
LIN {X 0,Y 594.267,Z 759.899,A -85,B 0,C 180,E1 -983.621,E2 -983.621} C_VEL
LIN {X 0,Y 594.296,Z 753.126,A -85,B 0,C 180,E1 -984.742,E2 -984.742} C_VEL
LIN {X 0,Y 594.351,Z 745.341,A -85,B 0,C 180,E1 -985.762,E2 -985.762} C_VEL
LIN {X 0,Y 594.372,Z 735.673,A -85,B 0,C 180,E1 -986.78,E2 -986.78} C_VEL
LIN {X 0,Y 594.453,Z 725.655,A -85,B 0,C 180,E1 -987.629,E2 -987.629} C_VEL
LIN {X 0,Y 594.464,Z 714.432,A -85,B 0,C 180,E1 -988.391,E2 -988.391} C_VEL
LIN {X 0,Y 594.538,Z 703.439,A -85,B 0,C 180,E1 -988.984,E2 -988.984} C_VEL
LIN {X 0,Y 594.575,Z 691.21,A -85,B 0,C 180,E1 -989.492,E2 -989.492} C_VEL
LIN {X 0,Y 594.613,Z 678.338,A -85,B 0,C 180,E1 -989.873,E2 -989.873} C_VEL
LIN {X 0,Y 594.683,Z 664.477,A -85,B 0,C 180,E1 -990.127,E2 -990.127} C_VEL
LIN {X 0,Y 594.598,Z 565.206,A -85,B 0,C 180,E1 -991.333,E2 -991.333} C_VEL
LIN {X 0,Y 594.374,Z 563.668,A -85,B 0,C 180,E1 -991.376,E2 -991.376} C_VEL
LIN {X 0,Y 594.392,Z 556.441,A -85,B 0,C 180,E1 -992.711,E2 -992.711} C_VEL
LIN {X 0,Y 594.392,Z 556.441,A -85,B 0,C 180,E1 -995.428,E2 -995.428} C_VEL
LIN {X 0,Y 594.385,Z 556.449,A -85,B 0,C 180,E1 -998.157,E2 -998.157} C_VEL
LIN {X 0,Y 594.389,Z 556.439,A -85,B 0,C 180,E1 -1001.072,E2 -1001.072} C_VEL
LIN {X 0,Y 594.387,Z 556.444,A -85,B 0,C 180,E1 -1003.678,E2 -1003.678} C_VEL
LIN {X 0,Y 594.396,Z 556.439,A -85,B 0,C 180,E1 -1006.719,E2 -1006.719} C_VEL
LIN {X 0,Y 594.369,Z 556.443,A -85,B 0,C 180,E1 -1009.334,E2 -1009.334} C_VEL
LIN {X 0,Y 594.37,Z 556.444,A -85,B 0,C 180,E1 -1011.503,E2 -1011.503} C_VEL
LIN {X 0,Y 594.39,Z 556.443,A -85,B 0,C 180,E1 -1014.445,E2 -1014.445} C_VEL
LIN {X 0,Y 594.383,Z 556.441,A -85,B 0,C 180,E1 -1016.699,E2 -1016.699} C_VEL
LIN {X 0,Y 594.381,Z 556.441,A -85,B 0,C 180,E1 -1018.998,E2 -1018.998} C_VEL
LIN {X 0,Y 594.391,Z 556.559,A -85,B 0,C 180,E1 -1021.422,E2 -1021.422} C_VEL
LIN {X 0,Y 594.365,Z 563.722,A -85,B 0,C 180,E1 -1022.723,E2 -1022.723} C_VEL
LIN {X 0,Y 594.752,Z 568.504,A -85,B 0,C 180,E1 -1022.8,E2 -1022.8} C_VEL
LIN {X 0,Y 594.663,Z 670.303,A -85,B 0,C 180,E1 -1024.051,E2 -1024.051} C_VEL
LIN {X 0,Y 594.609,Z 683.79,A -85,B 0,C 180,E1 -1024.361,E2 -1024.361} C_VEL
LIN {X 0,Y 594.551,Z 697.123,A -85,B 0,C 180,E1 -1024.825,E2 -1024.825} C_VEL
LIN {X 0,Y 594.513,Z 709.114,A -85,B 0,C 180,E1 -1025.397,E2 -1025.397} C_VEL
LIN {X 0,Y 594.459,Z 719.542,A -85,B 0,C 180,E1 -1026.026,E2 -1026.026} C_VEL
LIN {X 0,Y 594.418,Z 729.357,A -85,B 0,C 180,E1 -1026.756,E2 -1026.756} C_VEL
LIN {X 0,Y 594.376,Z 738.734,A -85,B 0,C 180,E1 -1027.606,E2 -1027.606} C_VEL
LIN {X 0,Y 594.322,Z 747.039,A -85,B 0,C 180,E1 -1028.534,E2 -1028.534} C_VEL
LIN {X 0,Y 594.306,Z 753.883,A -85,B 0,C 180,E1 -1029.465,E2 -1029.465} C_VEL
LIN {X 0,Y 594.268,Z 760.449,A -85,B 0,C 180,E1 -1030.574,E2 -1030.574} C_VEL
LIN {X 0,Y 594.245,Z 764.682,A -85,B 0,C 180,E1 -1031.474,E2 -1031.474} C_VEL
LIN {X 0,Y 594.268,Z 768.097,A -85,B 0,C 180,E1 -1032.383,E2 -1032.383} C_VEL
LIN {X 0,Y 594.248,Z 770.743,A -85,B 0,C 180,E1 -1033.309,E2 -1033.309} C_VEL
LIN {X 0,Y 594.225,Z 772.59,A -85,B 0,C 180,E1 -1034.25,E2 -1034.25} C_VEL
LIN {X 0,Y 594.226,Z 773.672,A -85,B 0,C 180,E1 -1035.203,E2 -1035.203} C_VEL
LIN {X 0,Y 594.232,Z 773.977,A -85,B 0,C 180,E1 -1036.173,E2 -1036.173} C_VEL
LIN {X 0,Y 594.245,Z 773.46,A -85,B 0,C 180,E1 -1037.159,E2 -1037.159} C_VEL
LIN {X 0,Y 594.222,Z 771.315,A -85,B 0,C 180,E1 -1038.522,E2 -1038.522} C_VEL
LIN {X 0,Y 594.248,Z 768.986,A -85,B 0,C 180,E1 -1039.423,E2 -1039.423} C_VEL
LIN {X 0,Y 594.239,Z 765.962,A -85,B 0,C 180,E1 -1040.308,E2 -1040.308} C_VEL
LIN {X 0,Y 594.288,Z 761.548,A -85,B 0,C 180,E1 -1041.305,E2 -1041.305} C_VEL
LIN {X 0,Y 594.269,Z 755.324,A -85,B 0,C 180,E1 -1042.405,E2 -1042.405} C_VEL
LIN {X 0,Y 594.316,Z 748.209,A -85,B 0,C 180,E1 -1043.409,E2 -1043.409} C_VEL
LIN {X 0,Y 594.355,Z 739.699,A -85,B 0,C 180,E1 -1044.383,E2 -1044.383} C_VEL
LIN {X 0,Y 594.395,Z 729.562,A -85,B 0,C 180,E1 -1045.318,E2 -1045.318} C_VEL
LIN {X 0,Y 594.466,Z 719.009,A -85,B 0,C 180,E1 -1046.1,E2 -1046.1} C_VEL
LIN {X 0,Y 594.53,Z 707.952,A -85,B 0,C 180,E1 -1046.756,E2 -1046.756} C_VEL
LIN {X 0,Y 594.563,Z 695.948,A -85,B 0,C 180,E1 -1047.313,E2 -1047.313} C_VEL
LIN {X 0,Y 594.618,Z 681.965,A -85,B 0,C 180,E1 -1047.78,E2 -1047.78} C_VEL
LIN {X 0,Y 594.675,Z 669.639,A -85,B 0,C 180,E1 -1048.049,E2 -1048.049} C_VEL
LIN {X 0,Y 594.714,Z 566.774,A -85,B 0,C 180,E1 -1049.312,E2 -1049.312} C_VEL
LIN {X 0,Y 594.326,Z 564.58,A -85,B 0,C 180,E1 -1049.363,E2 -1049.363} C_VEL
LIN {X 0,Y 594.4,Z 556.441,A -85,B 0,C 180,E1 -1051.104,E2 -1051.104} C_VEL
LIN {X 0,Y 594.369,Z 556.445,A -85,B 0,C 180,E1 -1054.055,E2 -1054.055} C_VEL
LIN {X 0,Y 594.388,Z 556.446,A -85,B 0,C 180,E1 -1056.296,E2 -1056.296} C_VEL
LIN {X 0,Y 594.399,Z 556.439,A -85,B 0,C 180,E1 -1059.224,E2 -1059.224} C_VEL
LIN {X 0,Y 594.378,Z 556.444,A -85,B 0,C 180,E1 -1062.096,E2 -1062.096} C_VEL
LIN {X 0,Y 594.365,Z 556.447,A -85,B 0,C 180,E1 -1064.219,E2 -1064.219} C_VEL
LIN {X 0,Y 594.367,Z 556.445,A -85,B 0,C 180,E1 -1067.017,E2 -1067.017} C_VEL
LIN {X 0,Y 594.391,Z 556.44,A -85,B 0,C 180,E1 -1069.784,E2 -1069.784} C_VEL
LIN {X 0,Y 594.411,Z 556.447,A -85,B 0,C 180,E1 -1072.527,E2 -1072.527} C_VEL
LIN {X 0,Y 594.4,Z 556.439,A -85,B 0,C 180,E1 -1075.252,E2 -1075.252} C_VEL
LIN {X 0,Y 594.387,Z 556.441,A -85,B 0,C 180,E1 -1077.967,E2 -1077.967} C_VEL
LIN {X 0,Y 594.419,Z 556.443,A -85,B 0,C 180,E1 -1080.677,E2 -1080.677} C_VEL
LIN {X 0,Y 594.376,Z 556.44,A -85,B 0,C 180,E1 -1083.389,E2 -1083.389} C_VEL
LIN {X 0,Y 594.382,Z 556.444,A -85,B 0,C 180,E1 -1086.109,E2 -1086.109} C_VEL
LIN {X 0,Y 594.395,Z 556.443,A -85,B 0,C 180,E1 -1088.842,E2 -1088.842} C_VEL
LIN {X 0,Y 594.387,Z 556.439,A -85,B 0,C 180,E1 -1091.596,E2 -1091.596} C_VEL
LIN {X 0,Y 594.381,Z 556.448,A -85,B 0,C 180,E1 -1094.377,E2 -1094.377} C_VEL
LIN {X 0,Y 594.384,Z 556.44,A -85,B 0,C 180,E1 -1097.194,E2 -1097.194} C_VEL
LIN {X 0,Y 594.375,Z 556.444,A -85,B 0,C 180,E1 -1100.054,E2 -1100.054} C_VEL
LIN {X 0,Y 594.391,Z 556.442,A -85,B 0,C 180,E1 -1102.966,E2 -1102.966} C_VEL
LIN {X 0,Y 594.373,Z 556.442,A -85,B 0,C 180,E1 -1105.193,E2 -1105.193} C_VEL
LIN {X 0,Y 594.376,Z 556.44,A -85,B 0,C 180,E1 -1107.527,E2 -1107.527} C_VEL
LIN {X 0,Y 594.393,Z 556.446,A -85,B 0,C 180,E1 -1110.332,E2 -1110.332} C_VEL
LIN {X 0,Y 594.373,Z 556.444,A -85,B 0,C 180,E1 -1112.951,E2 -1112.951} C_VEL
LIN {X 0,Y 594.375,Z 556.441,A -85,B 0,C 180,E1 -1115.407,E2 -1115.407} C_VEL
LIN {X 0,Y 594.386,Z 556.442,A -85,B 0,C 180,E1 -1117.941,E2 -1117.941} C_VEL
LIN {X 0,Y 594.384,Z 556.445,A -85,B 0,C 180,E1 -1120.824,E2 -1120.824} C_VEL
LIN {X 0,Y 594.382,Z 556.44,A -85,B 0,C 180,E1 -1123.298,E2 -1123.298} C_VEL
LIN {X 0,Y 594.363,Z 556.448,A -85,B 0,C 180,E1 -1126.161,E2 -1126.161} C_VEL
LIN {X 0,Y 594.378,Z 556.451,A -85,B 0,C 180,E1 -1128.537,E2 -1128.537} C_VEL
LIN {X 0,Y 594.383,Z 556.44,A -85,B 0,C 180,E1 -1131.296,E2 -1131.296} C_VEL
LIN {X 0,Y 594.349,Z 556.445,A -85,B 0,C 180,E1 -1133.756,E2 -1133.756} C_VEL
LIN {X 0,Y 594.38,Z 556.447,A -85,B 0,C 180,E1 -1136.24,E2 -1136.24} C_VEL
LIN {X 0,Y 594.368,Z 556.45,A -85,B 0,C 180,E1 -1138.651,E2 -1138.651} C_VEL
LIN {X 0,Y 594.383,Z 556.443,A -85,B 0,C 180,E1 -1141.043,E2 -1141.043} C_VEL
LIN {X 0,Y 594.388,Z 556.443,A -85,B 0,C 180,E1 -1143.977,E2 -1143.977} C_VEL
LIN {X 0,Y 594.387,Z 556.524,A -85,B 0,C 180,E1 -1145.136,E2 -1145.136} C_VEL
LIN {X 0,Y 594.97,Z 559.829,A -85,B 0,C 180,E1 -1145.58,E2 -1145.58} C_VEL
LIN {X 0,Y 594.853,Z 580.411,A -85,B 0,C 180,E1 -1148.152,E2 -1148.152} C_VEL
LIN {X 0,Y 594.684,Z 604.552,A -85,B 0,C 180,E1 -1151.11,E2 -1151.11} C_VEL
LIN {X 0,Y 594.563,Z 627.455,A -85,B 0,C 180,E1 -1153.873,E2 -1153.873} C_VEL
LIN {X 0,Y 594.51,Z 651.052,A -85,B 0,C 180,E1 -1156.659,E2 -1156.659} C_VEL
LIN {X 0,Y 594.758,Z 659.325,A -85,B 0,C 180,E1 -1156.765,E2 -1156.765} C_VEL
LIN {X 0,Y 594.678,Z 759.962,A -85,B 0,C 180,E1 -1157.999,E2 -1157.999} C_VEL
LIN {X 0,Y 594.642,Z 773.225,A -85,B 0,C 180,E1 -1158.301,E2 -1158.301} C_VEL
LIN {X 0,Y 594.591,Z 786.381,A -85,B 0,C 180,E1 -1158.75,E2 -1158.75} C_VEL
LIN {X 0,Y 594.538,Z 797.638,A -85,B 0,C 180,E1 -1159.27,E2 -1159.27} C_VEL
LIN {X 0,Y 594.472,Z 809.203,A -85,B 0,C 180,E1 -1159.958,E2 -1159.958} C_VEL
LIN {X 0,Y 594.413,Z 819.598,A -85,B 0,C 180,E1 -1160.73,E2 -1160.73} C_VEL
LIN {X 0,Y 594.383,Z 828.114,A -85,B 0,C 180,E1 -1161.501,E2 -1161.501} C_VEL
LIN {X 0,Y 594.347,Z 835.962,A -85,B 0,C 180,E1 -1162.356,E2 -1162.356} C_VEL
LIN {X 0,Y 594.282,Z 843.813,A -85,B 0,C 180,E1 -1163.408,E2 -1163.408} C_VEL
LIN {X 0,Y 594.289,Z 850.681,A -85,B 0,C 180,E1 -1164.571,E2 -1164.571} C_VEL
LIN {X 0,Y 594.271,Z 855.371,A -85,B 0,C 180,E1 -1165.591,E2 -1165.591} C_VEL
LIN {X 0,Y 594.268,Z 858.957,A -85,B 0,C 180,E1 -1166.61,E2 -1166.61} C_VEL
LIN {X 0,Y 594.226,Z 860.81,A -85,B 0,C 180,E1 -1167.288,E2 -1167.288} C_VEL
LIN {X 0,Y 594.239,Z 862.202,A -85,B 0,C 180,E1 -1167.967,E2 -1167.967} C_VEL
LIN {X 0,Y 594.239,Z 863.784,A -85,B 0,C 180,E1 -1169.322,E2 -1169.322} C_VEL
LIN {X 0,Y 594.236,Z 864,A -85,B 0,C 180,E1 -1170,E2 -1170} C_VEL
LIN {X 0,Y 594.247,Z 863.184,A -85,B 0,C 180,E1 -1171.355,E2 -1171.355} C_VEL
LIN {X 0,Y 594.239,Z 862.202,A -85,B 0,C 180,E1 -1172.033,E2 -1172.033} C_VEL
LIN {X 0,Y 594.226,Z 860.809,A -85,B 0,C 180,E1 -1172.712,E2 -1172.712} C_VEL
LIN {X 0,Y 594.289,Z 857.896,A -85,B 0,C 180,E1 -1173.729,E2 -1173.729} C_VEL
LIN {X 0,Y 594.241,Z 853.95,A -85,B 0,C 180,E1 -1174.749,E2 -1174.749} C_VEL
LIN {X 0,Y 594.304,Z 847.878,A -85,B 0,C 180,E1 -1175.939,E2 -1175.939} C_VEL
LIN {X 0,Y 594.308,Z 841.237,A -85,B 0,C 180,E1 -1176.962,E2 -1176.962} C_VEL
LIN {X 0,Y 594.359,Z 832.991,A -85,B 0,C 180,E1 -1177.986,E2 -1177.986} C_VEL
LIN {X 0,Y 594.382,Z 824.539,A -85,B 0,C 180,E1 -1178.842,E2 -1178.842} C_VEL
LIN {X 0,Y 594.423,Z 814.097,A -85,B 0,C 180,E1 -1179.699,E2 -1179.699} C_VEL
LIN {X 0,Y 594.489,Z 803.762,A -85,B 0,C 180,E1 -1180.386,E2 -1180.386} C_VEL
LIN {X 0,Y 594.56,Z 792.705,A -85,B 0,C 180,E1 -1180.974,E2 -1180.974} C_VEL
LIN {X 0,Y 594.602,Z 780.714,A -85,B 0,C 180,E1 -1181.464,E2 -1181.464} C_VEL
LIN {X 0,Y 594.641,Z 767.366,A -85,B 0,C 180,E1 -1181.85,E2 -1181.85} C_VEL
LIN {X 0,Y 594.687,Z 754.107,A -85,B 0,C 180,E1 -1182.087,E2 -1182.087} C_VEL
LIN {X 0,Y 594.648,Z 650.94,A -85,B 0,C 180,E1 -1183.339,E2 -1183.339} C_VEL
LIN {X 0,Y 594.494,Z 649.727,A -85,B 0,C 180,E1 -1183.371,E2 -1183.371} C_VEL
LIN {X 0,Y 594.612,Z 623.173,A -85,B 0,C 180,E1 -1186.126,E2 -1186.126} C_VEL
LIN {X 0,Y 594.768,Z 595.499,A -85,B 0,C 180,E1 -1189.036,E2 -1189.036} C_VEL
LIN {X 0,Y 594.966,Z 569.223,A -85,B 0,C 180,E1 -1191.844,E2 -1191.844} C_VEL
LIN {X 0,Y 594.955,Z 559.108,A -85,B 0,C 180,E1 -1192.943,E2 -1192.943} C_VEL
LIN {X 0,Y 594.38,Z 556.448,A -85,B 0,C 180,E1 -1193.288,E2 -1193.288} C_VEL
LIN {X 0,Y 594.393,Z 556.448,A -85,B 0,C 180,E1 -1196.024,E2 -1196.024} C_VEL
LIN {X 0,Y 594.383,Z 556.44,A -85,B 0,C 180,E1 -1198.998,E2 -1198.998} C_VEL
LIN {X 0,Y 594.384,Z 556.445,A -85,B 0,C 180,E1 -1201.643,E2 -1201.643} C_VEL
LIN {X 0,Y 594.394,Z 556.44,A -85,B 0,C 180,E1 -1204.578,E2 -1204.578} C_VEL
LIN {X 0,Y 594.382,Z 556.44,A -85,B 0,C 180,E1 -1207.086,E2 -1207.086} C_VEL
LIN {X 0,Y 594.376,Z 556.446,A -85,B 0,C 180,E1 -1209.774,E2 -1209.774} C_VEL
LIN {X 0,Y 594.365,Z 556.448,A -85,B 0,C 180,E1 -1212.374,E2 -1212.374} C_VEL
LIN {X 0,Y 594.358,Z 556.442,A -85,B 0,C 180,E1 -1215.19,E2 -1215.19} C_VEL
LIN {X 0,Y 594.367,Z 556.444,A -85,B 0,C 180,E1 -1217.624,E2 -1217.624} C_VEL
LIN {X 0,Y 594.391,Z 556.447,A -85,B 0,C 180,E1 -1220.321,E2 -1220.321} C_VEL
LIN {X 0,Y 594.383,Z 556.441,A -85,B 0,C 180,E1 -1222.913,E2 -1222.913} C_VEL
LIN {X 0,Y 594.378,Z 556.443,A -85,B 0,C 180,E1 -1225.86,E2 -1225.86} C_VEL
LIN {X 0,Y 594.384,Z 556.444,A -85,B 0,C 180,E1 -1228.65,E2 -1228.65} C_VEL
LIN {X 0,Y 594.376,Z 556.44,A -85,B 0,C 180,E1 -1231.041,E2 -1231.041} C_VEL
LIN {X 0,Y 594.388,Z 556.443,A -85,B 0,C 180,E1 -1233.974,E2 -1233.974} C_VEL
LIN {X 0,Y 594.386,Z 556.448,A -85,B 0,C 180,E1 -1236.296,E2 -1236.296} C_VEL
LIN {X 0,Y 594.398,Z 556.438,A -85,B 0,C 180,E1 -1239.224,E2 -1239.224} C_VEL
LIN {X 0,Y 594.374,Z 556.445,A -85,B 0,C 180,E1 -1242.096,E2 -1242.096} C_VEL
LIN {X 0,Y 594.362,Z 556.447,A -85,B 0,C 180,E1 -1244.219,E2 -1244.219} C_VEL
LIN {X 0,Y 594.363,Z 556.445,A -85,B 0,C 180,E1 -1247.017,E2 -1247.017} C_VEL
LIN {X 0,Y 594.39,Z 556.439,A -85,B 0,C 180,E1 -1249.784,E2 -1249.784} C_VEL
LIN {X 0,Y 594.394,Z 556.447,A -85,B 0,C 180,E1 -1252.527,E2 -1252.527} C_VEL
LIN {X 0,Y 594.401,Z 556.439,A -85,B 0,C 180,E1 -1255.252,E2 -1255.252} C_VEL
LIN {X 0,Y 594.387,Z 556.439,A -85,B 0,C 180,E1 -1257.967,E2 -1257.967} C_VEL
LIN {X 0,Y 594.425,Z 556.444,A -85,B 0,C 180,E1 -1260.677,E2 -1260.677} C_VEL
LIN {X 0,Y 594.376,Z 556.442,A -85,B 0,C 180,E1 -1263.389,E2 -1263.389} C_VEL
LIN {X 0,Y 594.38,Z 556.44,A -85,B 0,C 180,E1 -1266.109,E2 -1266.109} C_VEL
LIN {X 0,Y 594.395,Z 556.449,A -85,B 0,C 180,E1 -1268.842,E2 -1268.842} C_VEL
LIN {X 0,Y 594.386,Z 556.439,A -85,B 0,C 180,E1 -1271.596,E2 -1271.596} C_VEL
LIN {X 0,Y 594.379,Z 556.442,A -85,B 0,C 180,E1 -1274.377,E2 -1274.377} C_VEL
LIN {X 0,Y 594.354,Z 556.447,A -85,B 0,C 180,E1 -1275.342,E2 -1275.342} C_VEL
LIN {X 0,Y 593.686,Z 556.529,A -85,B 0,C 180,E1 -1275.908,E2 -1275.908} C_VEL
LIN {X 0,Y 590.833,Z 556.891,A -85,B 0,C 180,E1 -1276.826,E2 -1276.826} C_VEL
LIN {X 0,Y 588.427,Z 557.185,A -85,B 0,C 180,E1 -1277.565,E2 -1277.565} C_VEL
LIN {X 0,Y 587.399,Z 557.31,A -85,B 0,C 180,E1 -1278.135,E2 -1278.135} C_VEL
LIN {X 0,Y 587.318,Z 557.321,A -85,B 0,C 180,E1 -1278.328,E2 -1278.328} C_VEL
LIN {X 0,Y 587.348,Z 557.326,A -85,B 0,C 180,E1 -1281.045,E2 -1281.045} C_VEL
LIN {X 0,Y 587.331,Z 557.317,A -85,B 0,C 180,E1 -1284.007,E2 -1284.007} C_VEL
LIN {X 0,Y 587.355,Z 557.315,A -85,B 0,C 180,E1 -1286.278,E2 -1286.278} C_VEL
LIN {X 0,Y 587.343,Z 557.326,A -85,B 0,C 180,E1 -1289.135,E2 -1289.135} C_VEL
LIN {X 0,Y 587.347,Z 557.317,A -85,B 0,C 180,E1 -1291.838,E2 -1291.838} C_VEL
LIN {X 0,Y 587.347,Z 557.316,A -85,B 0,C 180,E1 -1294.35,E2 -1294.35} C_VEL
LIN {X 0,Y 587.347,Z 557.32,A -85,B 0,C 180,E1 -1296.747,E2 -1296.747} C_VEL
LIN {X 0,Y 587.341,Z 557.325,A -85,B 0,C 180,E1 -1299.36,E2 -1299.36} C_VEL
LIN {X 0,Y 587.329,Z 557.316,A -85,B 0,C 180,E1 -1302.109,E2 -1302.109} C_VEL
LIN {X 0,Y 587.311,Z 557.328,A -85,B 0,C 180,E1 -1305.09,E2 -1305.09} C_VEL
LIN {X 0,Y 587.319,Z 557.321,A -85,B 0,C 180,E1 -1307.926,E2 -1307.926} C_VEL
LIN {X 0,Y 587.342,Z 557.318,A -85,B 0,C 180,E1 -1310.642,E2 -1310.642} C_VEL
LIN {X 0,Y 587.351,Z 557.324,A -85,B 0,C 180,E1 -1313.293,E2 -1313.293} C_VEL
LIN {X 0,Y 587.365,Z 557.319,A -85,B 0,C 180,E1 -1315.781,E2 -1315.781} C_VEL
LIN {X 0,Y 587.341,Z 557.318,A -85,B 0,C 180,E1 -1318.232,E2 -1318.232} C_VEL
LIN {X 0,Y 587.349,Z 557.318,A -85,B 0,C 180,E1 -1320.867,E2 -1320.867} C_VEL
LIN {X 0,Y 587.314,Z 557.406,A -85,B 0,C 180,E1 -1323.05,E2 -1323.05} C_VEL
LIN {X 0,Y 587.301,Z 564.642,A -85,B 0,C 180,E1 -1324.577,E2 -1324.577} C_VEL
LIN {X 0,Y 587.861,Z 569.21,A -85,B 0,C 180,E1 -1324.651,E2 -1324.651} C_VEL
LIN {X 0,Y 587.72,Z 669.85,A -85,B 0,C 180,E1 -1325.899,E2 -1325.899} C_VEL
LIN {X 0,Y 587.648,Z 682.901,A -85,B 0,C 180,E1 -1326.195,E2 -1326.195} C_VEL
LIN {X 0,Y 587.598,Z 695.23,A -85,B 0,C 180,E1 -1326.614,E2 -1326.614} C_VEL
LIN {X 0,Y 587.539,Z 707.255,A -85,B 0,C 180,E1 -1327.166,E2 -1327.166} C_VEL
LIN {X 0,Y 587.444,Z 718.92,A -85,B 0,C 180,E1 -1327.861,E2 -1327.861} C_VEL
LIN {X 0,Y 587.373,Z 730.032,A -85,B 0,C 180,E1 -1328.698,E2 -1328.698} C_VEL
LIN {X 0,Y 587.333,Z 738.811,A -85,B 0,C 180,E1 -1329.513,E2 -1329.513} C_VEL
LIN {X 0,Y 587.279,Z 748.151,A -85,B 0,C 180,E1 -1330.584,E2 -1330.584} C_VEL
LIN {X 0,Y 587.247,Z 755.853,A -85,B 0,C 180,E1 -1331.691,E2 -1331.691} C_VEL
LIN {X 0,Y 587.189,Z 760.886,A -85,B 0,C 180,E1 -1332.59,E2 -1332.59} C_VEL
LIN {X 0,Y 587.162,Z 765.702,A -85,B 0,C 180,E1 -1333.664,E2 -1333.664} C_VEL
LIN {X 0,Y 587.164,Z 769.319,A -85,B 0,C 180,E1 -1334.733,E2 -1334.733} C_VEL
LIN {X 0,Y 587.16,Z 771.905,A -85,B 0,C 180,E1 -1335.82,E2 -1335.82} C_VEL
LIN {X 0,Y 587.145,Z 773.39,A -85,B 0,C 180,E1 -1336.855,E2 -1336.855} C_VEL
LIN {X 0,Y 587.16,Z 773.896,A -85,B 0,C 180,E1 -1337.558,E2 -1337.558} C_VEL
LIN {X 0,Y 587.165,Z 773.629,A -85,B 0,C 180,E1 -1338.959,E2 -1338.959} C_VEL
LIN {X 0,Y 587.143,Z 772.906,A -85,B 0,C 180,E1 -1339.657,E2 -1339.657} C_VEL
LIN {X 0,Y 587.152,Z 771.733,A -85,B 0,C 180,E1 -1340.353,E2 -1340.353} C_VEL
LIN {X 0,Y 587.151,Z 769.204,A -85,B 0,C 180,E1 -1341.395,E2 -1341.395} C_VEL
LIN {X 0,Y 587.188,Z 765.667,A -85,B 0,C 180,E1 -1342.435,E2 -1342.435} C_VEL
LIN {X 0,Y 587.175,Z 760.163,A -85,B 0,C 180,E1 -1343.639,E2 -1343.639} C_VEL
LIN {X 0,Y 587.208,Z 754.068,A -85,B 0,C 180,E1 -1344.678,E2 -1344.678} C_VEL
LIN {X 0,Y 587.296,Z 746.538,A -85,B 0,C 180,E1 -1345.711,E2 -1345.711} C_VEL
LIN {X 0,Y 587.305,Z 738.885,A -85,B 0,C 180,E1 -1346.57,E2 -1346.57} C_VEL
LIN {X 0,Y 587.393,Z 728.539,A -85,B 0,C 180,E1 -1347.514,E2 -1347.514} C_VEL
LIN {X 0,Y 587.459,Z 718.07,A -85,B 0,C 180,E1 -1348.286,E2 -1348.286} C_VEL
LIN {X 0,Y 587.505,Z 706.341,A -85,B 0,C 180,E1 -1348.972,E2 -1348.972} C_VEL
LIN {X 0,Y 587.604,Z 693.88,A -85,B 0,C 180,E1 -1349.529,E2 -1349.529} C_VEL
LIN {X 0,Y 587.682,Z 680.638,A -85,B 0,C 180,E1 -1349.957,E2 -1349.957} C_VEL
LIN {X 0,Y 587.746,Z 668.479,A -85,B 0,C 180,E1 -1350.214,E2 -1350.214} C_VEL
LIN {X 0,Y 587.743,Z 566.33,A -85,B 0,C 180,E1 -1351.477,E2 -1351.477} C_VEL
LIN {X 0,Y 587.328,Z 563.649,A -85,B 0,C 180,E1 -1351.543,E2 -1351.543} C_VEL
LIN {X 0,Y 587.36,Z 557.318,A -85,B 0,C 180,E1 -1352.743,E2 -1352.743} C_VEL
LIN {X 0,Y 587.357,Z 557.318,A -85,B 0,C 180,E1 -1355.493,E2 -1355.493} C_VEL
LIN {X 0,Y 587.345,Z 557.324,A -85,B 0,C 180,E1 -1358.255,E2 -1358.255} C_VEL
LIN {X 0,Y 587.352,Z 557.316,A -85,B 0,C 180,E1 -1361.133,E2 -1361.133} C_VEL
LIN {X 0,Y 587.368,Z 557.321,A -85,B 0,C 180,E1 -1364.26,E2 -1364.26} C_VEL
LIN {X 0,Y 587.357,Z 557.317,A -85,B 0,C 180,E1 -1367.405,E2 -1367.405} C_VEL
LIN {X 0,Y 587.33,Z 557.324,A -85,B 0,C 180,E1 -1370.304,E2 -1370.304} C_VEL
LIN {X 0,Y 587.317,Z 557.321,A -85,B 0,C 180,E1 -1373.258,E2 -1373.258} C_VEL
LIN {X 0,Y 587.334,Z 557.321,A -85,B 0,C 180,E1 -1375.516,E2 -1375.516} C_VEL
LIN {X 0,Y 587.35,Z 557.323,A -85,B 0,C 180,E1 -1377.817,E2 -1377.817} C_VEL
LIN {X 0,Y 587.346,Z 557.321,A -85,B 0,C 180,E1 -1380.511,E2 -1380.511} C_VEL
LIN {X 0,Y 587.364,Z 557.486,A -85,B 0,C 180,E1 -1381.415,E2 -1381.415} C_VEL
LIN {X 0,Y 587.324,Z 563.684,A -85,B 0,C 180,E1 -1382.554,E2 -1382.554} C_VEL
LIN {X 0,Y 587.84,Z 568.042,A -85,B 0,C 180,E1 -1382.636,E2 -1382.636} C_VEL
LIN {X 0,Y 587.735,Z 670.396,A -85,B 0,C 180,E1 -1383.91,E2 -1383.91} C_VEL
LIN {X 0,Y 587.656,Z 683.834,A -85,B 0,C 180,E1 -1384.222,E2 -1384.222} C_VEL
LIN {X 0,Y 587.591,Z 697.105,A -85,B 0,C 180,E1 -1384.69,E2 -1384.69} C_VEL
LIN {X 0,Y 587.552,Z 708.206,A -85,B 0,C 180,E1 -1385.22,E2 -1385.22} C_VEL
LIN {X 0,Y 587.419,Z 719.32,A -85,B 0,C 180,E1 -1385.89,E2 -1385.89} C_VEL
LIN {X 0,Y 587.392,Z 730.199,A -85,B 0,C 180,E1 -1386.713,E2 -1386.713} C_VEL
LIN {X 0,Y 587.314,Z 739.724,A -85,B 0,C 180,E1 -1387.609,E2 -1387.609} C_VEL
LIN {X 0,Y 587.258,Z 747.356,A -85,B 0,C 180,E1 -1388.484,E2 -1388.484} C_VEL
LIN {X 0,Y 587.227,Z 754.796,A -85,B 0,C 180,E1 -1389.526,E2 -1389.526} C_VEL
LIN {X 0,Y 587.177,Z 761.23,A -85,B 0,C 180,E1 -1390.66,E2 -1390.66} C_VEL
LIN {X 0,Y 587.167,Z 765.535,A -85,B 0,C 180,E1 -1391.627,E2 -1391.627} C_VEL
LIN {X 0,Y 587.164,Z 768.751,A -85,B 0,C 180,E1 -1392.551,E2 -1392.551} C_VEL
LIN {X 0,Y 587.149,Z 770.301,A -85,B 0,C 180,E1 -1393.101,E2 -1393.101} C_VEL
LIN {X 0,Y 587.15,Z 772.378,A -85,B 0,C 180,E1 -1394.095,E2 -1394.095} C_VEL
LIN {X 0,Y 587.148,Z 773.591,A -85,B 0,C 180,E1 -1395.072,E2 -1395.072} C_VEL
LIN {X 0,Y 587.131,Z 774,A -85,B 0,C 180,E1 -1396.031,E2 -1396.031} C_VEL
LIN {X 0,Y 587.16,Z 773.617,A -85,B 0,C 180,E1 -1396.979,E2 -1396.979} C_VEL
LIN {X 0,Y 587.157,Z 772.514,A -85,B 0,C 180,E1 -1397.91,E2 -1397.91} C_VEL
LIN {X 0,Y 587.127,Z 770.411,A -85,B 0,C 180,E1 -1398.947,E2 -1398.947} C_VEL
LIN {X 0,Y 587.17,Z 766.148,A -85,B 0,C 180,E1 -1400.311,E2 -1400.311} C_VEL
LIN {X 0,Y 587.178,Z 760.824,A -85,B 0,C 180,E1 -1401.509,E2 -1401.509} C_VEL
LIN {X 0,Y 587.216,Z 754.571,A -85,B 0,C 180,E1 -1402.599,E2 -1402.599} C_VEL
LIN {X 0,Y 587.26,Z 746.83,A -85,B 0,C 180,E1 -1403.673,E2 -1403.673} C_VEL
LIN {X 0,Y 587.329,Z 738.662,A -85,B 0,C 180,E1 -1404.593,E2 -1404.593} C_VEL
LIN {X 0,Y 587.388,Z 728.265,A -85,B 0,C 180,E1 -1405.536,E2 -1405.536} C_VEL
LIN {X 0,Y 587.482,Z 717.744,A -85,B 0,C 180,E1 -1406.304,E2 -1406.304} C_VEL
LIN {X 0,Y 587.533,Z 707.167,A -85,B 0,C 180,E1 -1406.928,E2 -1406.928} C_VEL
LIN {X 0,Y 587.62,Z 695.004,A -85,B 0,C 180,E1 -1407.485,E2 -1407.485} C_VEL
LIN {X 0,Y 587.681,Z 681.624,A -85,B 0,C 180,E1 -1407.93,E2 -1407.93} C_VEL
LIN {X 0,Y 587.727,Z 669.131,A -85,B 0,C 180,E1 -1408.201,E2 -1408.201} C_VEL
LIN {X 0,Y 587.698,Z 567.174,A -85,B 0,C 180,E1 -1409.468,E2 -1409.468} C_VEL
LIN {X 0,Y 587.285,Z 564.576,A -85,B 0,C 180,E1 -1409.527,E2 -1409.527} C_VEL
LIN {X 0,Y 587.351,Z 557.32,A -85,B 0,C 180,E1 -1411.07,E2 -1411.07} C_VEL
LIN {X 0,Y 587.353,Z 557.317,A -85,B 0,C 180,E1 -1413.818,E2 -1413.818} C_VEL
LIN {X 0,Y 587.332,Z 557.321,A -85,B 0,C 180,E1 -1415.993,E2 -1415.993} C_VEL
LIN {X 0,Y 587.338,Z 557.322,A -85,B 0,C 180,E1 -1418.963,E2 -1418.963} C_VEL
LIN {X 0,Y 587.324,Z 557.321,A -85,B 0,C 180,E1 -1421.873,E2 -1421.873} C_VEL
LIN {X 0,Y 587.321,Z 557.322,A -85,B 0,C 180,E1 -1424.025,E2 -1424.025} C_VEL
LIN {X 0,Y 587.353,Z 557.32,A -85,B 0,C 180,E1 -1426.154,E2 -1426.154} C_VEL
LIN {X 0,Y 587.338,Z 557.321,A -85,B 0,C 180,E1 -1428.962,E2 -1428.962} C_VEL
LIN {X 0,Y 587.365,Z 557.315,A -85,B 0,C 180,E1 -1431.745,E2 -1431.745} C_VEL
LIN {X 0,Y 587.354,Z 557.326,A -85,B 0,C 180,E1 -1434.507,E2 -1434.507} C_VEL
LIN {X 0,Y 587.376,Z 557.313,A -85,B 0,C 180,E1 -1437.257,E2 -1437.257} C_VEL
LIN {X 0,Y 587.372,Z 557.316,A -85,B 0,C 180,E1 -1440,E2 -1440} C_VEL
LIN {X 0,Y 587.375,Z 557.319,A -85,B 0,C 180,E1 -1442.743,E2 -1442.743} C_VEL
LIN {X 0,Y 587.355,Z 557.315,A -85,B 0,C 180,E1 -1445.493,E2 -1445.493} C_VEL
LIN {X 0,Y 587.366,Z 557.32,A -85,B 0,C 180,E1 -1448.255,E2 -1448.255} C_VEL
LIN {X 0,Y 587.351,Z 557.317,A -85,B 0,C 180,E1 -1451.142,E2 -1451.142} C_VEL
LIN {X 0,Y 587.355,Z 557.321,A -85,B 0,C 180,E1 -1454.261,E2 -1454.261} C_VEL
LIN {X 0,Y 587.351,Z 557.315,A -85,B 0,C 180,E1 -1457.406,E2 -1457.406} C_VEL
LIN {X 0,Y 587.33,Z 557.325,A -85,B 0,C 180,E1 -1460.305,E2 -1460.305} C_VEL
LIN {X 0,Y 587.36,Z 557.315,A -85,B 0,C 180,E1 -1463.257,E2 -1463.257} C_VEL
LIN {X 0,Y 587.356,Z 557.322,A -85,B 0,C 180,E1 -1466.278,E2 -1466.278} C_VEL
LIN {X 0,Y 587.346,Z 557.318,A -85,B 0,C 180,E1 -1469.135,E2 -1469.135} C_VEL
LIN {X 0,Y 587.351,Z 557.317,A -85,B 0,C 180,E1 -1471.839,E2 -1471.839} C_VEL
LIN {X 0,Y 587.35,Z 557.324,A -85,B 0,C 180,E1 -1474.35,E2 -1474.35} C_VEL
LIN {X 0,Y 587.347,Z 557.323,A -85,B 0,C 180,E1 -1476.747,E2 -1476.747} C_VEL
LIN {X 0,Y 587.343,Z 557.317,A -85,B 0,C 180,E1 -1479.36,E2 -1479.36} C_VEL
LIN {X 0,Y 587.333,Z 557.322,A -85,B 0,C 180,E1 -1482.109,E2 -1482.109} C_VEL
LIN {X 0,Y 587.311,Z 557.323,A -85,B 0,C 180,E1 -1485.09,E2 -1485.09} C_VEL
LIN {X 0,Y 587.349,Z 557.319,A -85,B 0,C 180,E1 -1487.928,E2 -1487.928} C_VEL
LIN {X 0,Y 587.33,Z 557.321,A -85,B 0,C 180,E1 -1491.059,E2 -1491.059} C_VEL
LIN {X 0,Y 587.344,Z 557.317,A -85,B 0,C 180,E1 -1493.293,E2 -1493.293} C_VEL
LIN {X 0,Y 587.365,Z 557.315,A -85,B 0,C 180,E1 -1495.781,E2 -1495.781} C_VEL
LIN {X 0,Y 587.341,Z 557.324,A -85,B 0,C 180,E1 -1498.232,E2 -1498.232} C_VEL
LIN {X 0,Y 587.349,Z 557.321,A -85,B 0,C 180,E1 -1500.867,E2 -1500.867} C_VEL
LIN {X 0,Y 587.361,Z 557.318,A -85,B 0,C 180,E1 -1503.819,E2 -1503.819} C_VEL
LIN {X 0,Y 587.358,Z 557.44,A -85,B 0,C 180,E1 -1504.935,E2 -1504.935} C_VEL
LIN {X 0,Y 588.094,Z 561.11,A -85,B 0,C 180,E1 -1505.44,E2 -1505.44} C_VEL
LIN {X 0,Y 587.987,Z 578.941,A -85,B 0,C 180,E1 -1507.698,E2 -1507.698} C_VEL
LIN {X 0,Y 587.763,Z 602.066,A -85,B 0,C 180,E1 -1510.573,E2 -1510.573} C_VEL
LIN {X 0,Y 587.612,Z 624.515,A -85,B 0,C 180,E1 -1513.319,E2 -1513.319} C_VEL
LIN {X 0,Y 587.504,Z 648.037,A -85,B 0,C 180,E1 -1516.158,E2 -1516.158} C_VEL
LIN {X 0,Y 587.491,Z 650.794,A -85,B 0,C 180,E1 -1516.488,E2 -1516.488} C_VEL
LIN {X 0,Y 587.863,Z 657.536,A -85,B 0,C 180,E1 -1516.585,E2 -1516.585} C_VEL
LIN {X 0,Y 587.737,Z 759.962,A -85,B 0,C 180,E1 -1517.856,E2 -1517.856} C_VEL
LIN {X 0,Y 587.702,Z 772.465,A -85,B 0,C 180,E1 -1518.139,E2 -1518.139} C_VEL
LIN {X 0,Y 587.61,Z 784.594,A -85,B 0,C 180,E1 -1518.545,E2 -1518.545} C_VEL
LIN {X 0,Y 587.542,Z 795.932,A -85,B 0,C 180,E1 -1519.054,E2 -1519.054} C_VEL
LIN {X 0,Y 587.471,Z 806.587,A -85,B 0,C 180,E1 -1519.663,E2 -1519.663} C_VEL
LIN {X 0,Y 587.39,Z 817.478,A -85,B 0,C 180,E1 -1520.444,E2 -1520.444} C_VEL
LIN {X 0,Y 587.321,Z 828.114,A -85,B 0,C 180,E1 -1521.398,E2 -1521.398} C_VEL
LIN {X 0,Y 587.273,Z 835.962,A -85,B 0,C 180,E1 -1522.263,E2 -1522.263} C_VEL
LIN {X 0,Y 587.23,Z 842.471,A -85,B 0,C 180,E1 -1523.127,E2 -1523.127} C_VEL
LIN {X 0,Y 587.236,Z 848.867,A -85,B 0,C 180,E1 -1524.161,E2 -1524.161} C_VEL
LIN {X 0,Y 587.147,Z 853.95,A -85,B 0,C 180,E1 -1525.194,E2 -1525.194} C_VEL
LIN {X 0,Y 587.213,Z 857.896,A -85,B 0,C 180,E1 -1526.226,E2 -1526.226} C_VEL
LIN {X 0,Y 587.132,Z 860.81,A -85,B 0,C 180,E1 -1527.256,E2 -1527.256} C_VEL
LIN {X 0,Y 587.138,Z 862.201,A -85,B 0,C 180,E1 -1527.942,E2 -1527.942} C_VEL
LIN {X 0,Y 587.14,Z 863.784,A -85,B 0,C 180,E1 -1529.314,E2 -1529.314} C_VEL
LIN {X 0,Y 587.137,Z 864,A -85,B 0,C 180,E1 -1530,E2 -1530} C_VEL
LIN {X 0,Y 587.147,Z 863.185,A -85,B 0,C 180,E1 -1531.372,E2 -1531.372} C_VEL
LIN {X 0,Y 587.138,Z 862.201,A -85,B 0,C 180,E1 -1532.058,E2 -1532.058} C_VEL
LIN {X 0,Y 587.132,Z 860.809,A -85,B 0,C 180,E1 -1532.744,E2 -1532.744} C_VEL
LIN {X 0,Y 587.213,Z 857.896,A -85,B 0,C 180,E1 -1533.774,E2 -1533.774} C_VEL
LIN {X 0,Y 587.147,Z 853.95,A -85,B 0,C 180,E1 -1534.806,E2 -1534.806} C_VEL
LIN {X 0,Y 587.217,Z 847.878,A -85,B 0,C 180,E1 -1536.011,E2 -1536.011} C_VEL
LIN {X 0,Y 587.245,Z 841.238,A -85,B 0,C 180,E1 -1537.046,E2 -1537.046} C_VEL
LIN {X 0,Y 587.299,Z 832.992,A -85,B 0,C 180,E1 -1538.083,E2 -1538.083} C_VEL
LIN {X 0,Y 587.343,Z 824.54,A -85,B 0,C 180,E1 -1538.949,E2 -1538.949} C_VEL
LIN {X 0,Y 587.411,Z 814.098,A -85,B 0,C 180,E1 -1539.816,E2 -1539.816} C_VEL
LIN {X 0,Y 587.507,Z 803.762,A -85,B 0,C 180,E1 -1540.511,E2 -1540.511} C_VEL
LIN {X 0,Y 587.583,Z 791.809,A -85,B 0,C 180,E1 -1541.149,E2 -1541.149} C_VEL
LIN {X 0,Y 587.657,Z 779.603,A -85,B 0,C 180,E1 -1541.639,E2 -1541.639} C_VEL
LIN {X 0,Y 587.68,Z 766.452,A -85,B 0,C 180,E1 -1542.014,E2 -1542.014} C_VEL
LIN {X 0,Y 587.768,Z 754.107,A -85,B 0,C 180,E1 -1542.231,E2 -1542.231} C_VEL
LIN {X 0,Y 587.792,Z 652.17,A -85,B 0,C 180,E1 -1543.482,E2 -1543.482} C_VEL
LIN {X 0,Y 587.512,Z 649.727,A -85,B 0,C 180,E1 -1543.533,E2 -1543.533} C_VEL
LIN {X 0,Y 587.675,Z 621.487,A -85,B 0,C 180,E1 -1546.5,E2 -1546.5} C_VEL
LIN {X 0,Y 587.872,Z 595.17,A -85,B 0,C 180,E1 -1549.304,E2 -1549.304} C_VEL
LIN {X 0,Y 588.113,Z 569.223,A -85,B 0,C 180,E1 -1552.112,E2 -1552.112} C_VEL
LIN {X 0,Y 588.097,Z 560.728,A -85,B 0,C 180,E1 -1553.047,E2 -1553.047} C_VEL
LIN {X 0,Y 587.348,Z 557.325,A -85,B 0,C 180,E1 -1553.467,E2 -1553.467} C_VEL
LIN {X 0,Y 587.364,Z 557.319,A -85,B 0,C 180,E1 -1556.277,E2 -1556.277} C_VEL
LIN {X 0,Y 587.351,Z 557.317,A -85,B 0,C 180,E1 -1559.133,E2 -1559.133} C_VEL
LIN {X 0,Y 587.349,Z 557.325,A -85,B 0,C 180,E1 -1561.836,E2 -1561.836} C_VEL
LIN {X 0,Y 587.356,Z 557.32,A -85,B 0,C 180,E1 -1564.348,E2 -1564.348} C_VEL
LIN {X 0,Y 587.35,Z 557.317,A -85,B 0,C 180,E1 -1566.746,E2 -1566.746} C_VEL
LIN {X 0,Y 587.344,Z 557.317,A -85,B 0,C 180,E1 -1569.358,E2 -1569.358} C_VEL
LIN {X 0,Y 587.33,Z 557.328,A -85,B 0,C 180,E1 -1572.107,E2 -1572.107} C_VEL
LIN {X 0,Y 587.311,Z 557.321,A -85,B 0,C 180,E1 -1574.91,E2 -1574.91} C_VEL
LIN {X 0,Y 587.318,Z 557.32,A -85,B 0,C 180,E1 -1576.994,E2 -1576.994} C_VEL
LIN {X 0,Y 587.325,Z 557.322,A -85,B 0,C 180,E1 -1579.746,E2 -1579.746} C_VEL
LIN {X 0,Y 587.343,Z 557.325,A -85,B 0,C 180,E1 -1582.392,E2 -1582.392} C_VEL
LIN {X 0,Y 587.341,Z 557.317,A -85,B 0,C 180,E1 -1584.945,E2 -1584.945} C_VEL
LIN {X 0,Y 587.332,Z 557.318,A -85,B 0,C 180,E1 -1587.42,E2 -1587.42} C_VEL
LIN {X 0,Y 587.34,Z 557.32,A -85,B 0,C 180,E1 -1589.83,E2 -1589.83} C_VEL
LIN {X 0,Y 587.343,Z 557.326,A -85,B 0,C 180,E1 -1592.306,E2 -1592.306} C_VEL
LIN {X 0,Y 587.335,Z 557.327,A -85,B 0,C 180,E1 -1594.483,E2 -1594.483} C_VEL
LIN {X 0,Y 587.331,Z 557.316,A -85,B 0,C 180,E1 -1597.486,E2 -1597.486} C_VEL
LIN {X 0,Y 587.325,Z 557.319,A -85,B 0,C 180,E1 -1599.695,E2 -1599.695} C_VEL
LIN {X 0,Y 587.35,Z 557.324,A -85,B 0,C 180,E1 -1602.594,E2 -1602.594} C_VEL
LIN {X 0,Y 587.354,Z 557.315,A -85,B 0,C 180,E1 -1605.739,E2 -1605.739} C_VEL
LIN {X 0,Y 587.351,Z 557.321,A -85,B 0,C 180,E1 -1608.858,E2 -1608.858} C_VEL
LIN {X 0,Y 587.364,Z 557.313,A -85,B 0,C 180,E1 -1611.745,E2 -1611.745} C_VEL
LIN {X 0,Y 587.359,Z 557.323,A -85,B 0,C 180,E1 -1614.507,E2 -1614.507} C_VEL
LIN {X 0,Y 587.376,Z 557.313,A -85,B 0,C 180,E1 -1617.257,E2 -1617.257} C_VEL
LIN {X 0,Y 587.372,Z 557.313,A -85,B 0,C 180,E1 -1620,E2 -1620} C_VEL
LIN {X 0,Y 587.375,Z 557.324,A -85,B 0,C 180,E1 -1622.743,E2 -1622.743} C_VEL
LIN {X 0,Y 587.356,Z 557.314,A -85,B 0,C 180,E1 -1625.493,E2 -1625.493} C_VEL
LIN {X 0,Y 587.364,Z 557.316,A -85,B 0,C 180,E1 -1628.255,E2 -1628.255} C_VEL
LIN {X 0,Y 587.351,Z 557.32,A -85,B 0,C 180,E1 -1631.142,E2 -1631.142} C_VEL
LIN {X 0,Y 587.354,Z 557.316,A -85,B 0,C 180,E1 -1634.261,E2 -1634.261} C_VEL
LIN {X 0,Y 587.351,Z 557.318,A -85,B 0,C 180,E1 -1637.406,E2 -1637.406} C_VEL
LIN {X 0,Y 587.318,Z 557.321,A -85,B 0,C 180,E1 -1638.328,E2 -1638.328} C_VEL
LIN {X 0,Y 586.664,Z 557.41,A -85,B 0,C 180,E1 -1638.9,E2 -1638.9} C_VEL
LIN {X 0,Y 583.834,Z 557.766,A -85,B 0,C 180,E1 -1639.828,E2 -1639.828} C_VEL
LIN {X 0,Y 581.424,Z 558.066,A -85,B 0,C 180,E1 -1640.575,E2 -1640.575} C_VEL
LIN {X 0,Y 580.372,Z 558.193,A -85,B 0,C 180,E1 -1641.152,E2 -1641.152} C_VEL
LIN {X 0,Y 580.277,Z 558.202,A -85,B 0,C 180,E1 -1641.347,E2 -1641.347} C_VEL
LIN {X 0,Y 580.293,Z 558.195,A -85,B 0,C 180,E1 -1644.317,E2 -1644.317} C_VEL
LIN {X 0,Y 580.303,Z 558.197,A -85,B 0,C 180,E1 -1646.622,E2 -1646.622} C_VEL
LIN {X 0,Y 580.298,Z 558.2,A -85,B 0,C 180,E1 -1649.311,E2 -1649.311} C_VEL
LIN {X 0,Y 580.295,Z 558.195,A -85,B 0,C 180,E1 -1652.201,E2 -1652.201} C_VEL
LIN {X 0,Y 580.293,Z 558.197,A -85,B 0,C 180,E1 -1654.696,E2 -1654.696} C_VEL
LIN {X 0,Y 580.296,Z 558.204,A -85,B 0,C 180,E1 -1657.269,E2 -1657.269} C_VEL
LIN {X 0,Y 580.293,Z 558.194,A -85,B 0,C 180,E1 -1660.272,E2 -1660.272} C_VEL
LIN {X 0,Y 580.277,Z 558.196,A -85,B 0,C 180,E1 -1662.707,E2 -1662.707} C_VEL
LIN {X 0,Y 580.265,Z 558.204,A -85,B 0,C 180,E1 -1665.61,E2 -1665.61} C_VEL
LIN {X 0,Y 580.276,Z 558.196,A -85,B 0,C 180,E1 -1668.232,E2 -1668.232} C_VEL
LIN {X 0,Y 580.285,Z 558.2,A -85,B 0,C 180,E1 -1670.967,E2 -1670.967} C_VEL
LIN {X 0,Y 580.294,Z 558.202,A -85,B 0,C 180,E1 -1673.599,E2 -1673.599} C_VEL
LIN {X 0,Y 580.318,Z 558.193,A -85,B 0,C 180,E1 -1676.146,E2 -1676.146} C_VEL
LIN {X 0,Y 580.275,Z 558.198,A -85,B 0,C 180,E1 -1678.615,E2 -1678.615} C_VEL
LIN {X 0,Y 580.293,Z 558.198,A -85,B 0,C 180,E1 -1681.025,E2 -1681.025} C_VEL
LIN {X 0,Y 580.256,Z 558.212,A -85,B 0,C 180,E1 -1683.036,E2 -1683.036} C_VEL
LIN {X 0,Y 580.275,Z 564.635,A -85,B 0,C 180,E1 -1684.41,E2 -1684.41} C_VEL
LIN {X 0,Y 580.983,Z 569.841,A -85,B 0,C 180,E1 -1684.497,E2 -1684.497} C_VEL
LIN {X 0,Y 580.796,Z 669.973,A -85,B 0,C 180,E1 -1685.754,E2 -1685.754} C_VEL
LIN {X 0,Y 580.692,Z 683.148,A -85,B 0,C 180,E1 -1686.058,E2 -1686.058} C_VEL
LIN {X 0,Y 580.658,Z 694.828,A -85,B 0,C 180,E1 -1686.459,E2 -1686.459} C_VEL
LIN {X 0,Y 580.551,Z 707.414,A -85,B 0,C 180,E1 -1687.042,E2 -1687.042} C_VEL
LIN {X 0,Y 580.433,Z 719.358,A -85,B 0,C 180,E1 -1687.767,E2 -1687.767} C_VEL
LIN {X 0,Y 580.352,Z 730.269,A -85,B 0,C 180,E1 -1688.605,E2 -1688.605} C_VEL
LIN {X 0,Y 580.282,Z 739.098,A -85,B 0,C 180,E1 -1689.438,E2 -1689.438} C_VEL
LIN {X 0,Y 580.194,Z 747.255,A -85,B 0,C 180,E1 -1690.377,E2 -1690.377} C_VEL
LIN {X 0,Y 580.155,Z 754.888,A -85,B 0,C 180,E1 -1691.459,E2 -1691.459} C_VEL
LIN {X 0,Y 580.109,Z 760.099,A -85,B 0,C 180,E1 -1692.37,E2 -1692.37} C_VEL
LIN {X 0,Y 580.082,Z 765.213,A -85,B 0,C 180,E1 -1693.488,E2 -1693.488} C_VEL
LIN {X 0,Y 580.09,Z 768.867,A -85,B 0,C 180,E1 -1694.542,E2 -1694.542} C_VEL
LIN {X 0,Y 580.067,Z 771.836,A -85,B 0,C 180,E1 -1695.759,E2 -1695.759} C_VEL
LIN {X 0,Y 580.06,Z 773.223,A -85,B 0,C 180,E1 -1696.691,E2 -1696.691} C_VEL
LIN {X 0,Y 580.05,Z 773.819,A -85,B 0,C 180,E1 -1697.403,E2 -1697.403} C_VEL
LIN {X 0,Y 580.053,Z 773.991,A -85,B 0,C 180,E1 -1698.114,E2 -1698.114} C_VEL
LIN {X 0,Y 580.072,Z 773.659,A -85,B 0,C 180,E1 -1698.925,E2 -1698.925} C_VEL
LIN {X 0,Y 580.059,Z 772.027,A -85,B 0,C 180,E1 -1700.234,E2 -1700.234} C_VEL
LIN {X 0,Y 580.031,Z 770.519,A -85,B 0,C 180,E1 -1700.938,E2 -1700.938} C_VEL
LIN {X 0,Y 580.082,Z 767.466,A -85,B 0,C 180,E1 -1701.991,E2 -1701.991} C_VEL
LIN {X 0,Y 580.139,Z 763.363,A -85,B 0,C 180,E1 -1703.042,E2 -1703.042} C_VEL
LIN {X 0,Y 580.161,Z 757.104,A -85,B 0,C 180,E1 -1704.264,E2 -1704.264} C_VEL
LIN {X 0,Y 580.194,Z 750.305,A -85,B 0,C 180,E1 -1705.31,E2 -1705.31} C_VEL
LIN {X 0,Y 580.223,Z 741.86,A -85,B 0,C 180,E1 -1706.354,E2 -1706.354} C_VEL
LIN {X 0,Y 580.317,Z 733.219,A -85,B 0,C 180,E1 -1707.223,E2 -1707.223} C_VEL
LIN {X 0,Y 580.399,Z 722.643,A -85,B 0,C 180,E1 -1708.092,E2 -1708.092} C_VEL
LIN {X 0,Y 580.467,Z 712.095,A -85,B 0,C 180,E1 -1708.786,E2 -1708.786} C_VEL
LIN {X 0,Y 580.629,Z 700.397,A -85,B 0,C 180,E1 -1709.393,E2 -1709.393} C_VEL
LIN {X 0,Y 580.694,Z 688.318,A -85,B 0,C 180,E1 -1709.87,E2 -1709.87} C_VEL
LIN {X 0,Y 580.75,Z 675.965,A -85,B 0,C 180,E1 -1710.217,E2 -1710.217} C_VEL
LIN {X 0,Y 580.832,Z 661.683,A -85,B 0,C 180,E1 -1710.455,E2 -1710.455} C_VEL
LIN {X 0,Y 580.9,Z 567.44,A -85,B 0,C 180,E1 -1711.625,E2 -1711.625} C_VEL
LIN {X 0,Y 580.269,Z 563.748,A -85,B 0,C 180,E1 -1711.692,E2 -1711.692} C_VEL
LIN {X 0,Y 580.325,Z 558.195,A -85,B 0,C 180,E1 -1712.733,E2 -1712.733} C_VEL
LIN {X 0,Y 580.323,Z 558.195,A -85,B 0,C 180,E1 -1715.56,E2 -1715.56} C_VEL
LIN {X 0,Y 580.327,Z 558.195,A -85,B 0,C 180,E1 -1717.655,E2 -1717.655} C_VEL
LIN {X 0,Y 580.298,Z 558.198,A -85,B 0,C 180,E1 -1720.466,E2 -1720.466} C_VEL
LIN {X 0,Y 580.306,Z 558.196,A -85,B 0,C 180,E1 -1722.591,E2 -1722.591} C_VEL
LIN {X 0,Y 580.289,Z 558.197,A -85,B 0,C 180,E1 -1724.734,E2 -1724.734} C_VEL
LIN {X 0,Y 580.302,Z 558.198,A -85,B 0,C 180,E1 -1727.624,E2 -1727.624} C_VEL
LIN {X 0,Y 580.306,Z 558.2,A -85,B 0,C 180,E1 -1729.822,E2 -1729.822} C_VEL
LIN {X 0,Y 580.292,Z 558.196,A -85,B 0,C 180,E1 -1732.802,E2 -1732.802} C_VEL
LIN {X 0,Y 580.307,Z 558.194,A -85,B 0,C 180,E1 -1735.079,E2 -1735.079} C_VEL
LIN {X 0,Y 580.302,Z 558.203,A -85,B 0,C 180,E1 -1738.185,E2 -1738.185} C_VEL
LIN {X 0,Y 580.322,Z 558.194,A -85,B 0,C 180,E1 -1741.278,E2 -1741.278} C_VEL
LIN {X 0,Y 580.309,Z 558.289,A -85,B 0,C 180,E1 -1741.383,E2 -1741.383} C_VEL
LIN {X 0,Y 580.293,Z 563.795,A -85,B 0,C 180,E1 -1742.405,E2 -1742.405} C_VEL
LIN {X 0,Y 580.948,Z 568.513,A -85,B 0,C 180,E1 -1742.48,E2 -1742.48} C_VEL
LIN {X 0,Y 580.792,Z 670.146,A -85,B 0,C 180,E1 -1743.759,E2 -1743.759} C_VEL
LIN {X 0,Y 580.729,Z 683.238,A -85,B 0,C 180,E1 -1744.061,E2 -1744.061} C_VEL
LIN {X 0,Y 580.651,Z 696.614,A -85,B 0,C 180,E1 -1744.531,E2 -1744.531} C_VEL
LIN {X 0,Y 580.58,Z 708.37,A -85,B 0,C 180,E1 -1745.098,E2 -1745.098} C_VEL
LIN {X 0,Y 580.415,Z 719.505,A -85,B 0,C 180,E1 -1745.779,E2 -1745.779} C_VEL
LIN {X 0,Y 580.362,Z 730.081,A -85,B 0,C 180,E1 -1746.589,E2 -1746.589} C_VEL
LIN {X 0,Y 580.258,Z 740.583,A -85,B 0,C 180,E1 -1747.598,E2 -1747.598} C_VEL
LIN {X 0,Y 580.18,Z 748.922,A -85,B 0,C 180,E1 -1748.596,E2 -1748.596} C_VEL
LIN {X 0,Y 580.157,Z 755.313,A -85,B 0,C 180,E1 -1749.531,E2 -1749.531} C_VEL
LIN {X 0,Y 580.108,Z 760.897,A -85,B 0,C 180,E1 -1750.53,E2 -1750.53} C_VEL
LIN {X 0,Y 580.099,Z 766.356,A -85,B 0,C 180,E1 -1751.783,E2 -1751.783} C_VEL
LIN {X 0,Y 580.073,Z 769.403,A -85,B 0,C 180,E1 -1752.724,E2 -1752.724} C_VEL
LIN {X 0,Y 580.024,Z 771.669,A -85,B 0,C 180,E1 -1753.681,E2 -1753.681} C_VEL
LIN {X 0,Y 580.035,Z 773.172,A -85,B 0,C 180,E1 -1754.647,E2 -1754.647} C_VEL
LIN {X 0,Y 580.036,Z 773.904,A -85,B 0,C 180,E1 -1755.631,E2 -1755.631} C_VEL
LIN {X 0,Y 580.026,Z 773.829,A -85,B 0,C 180,E1 -1756.634,E2 -1756.634} C_VEL
LIN {X 0,Y 580.058,Z 772.91,A -85,B 0,C 180,E1 -1757.651,E2 -1757.651} C_VEL
LIN {X 0,Y 580.037,Z 771.067,A -85,B 0,C 180,E1 -1758.695,E2 -1758.695} C_VEL
LIN {X 0,Y 580.086,Z 767.267,A -85,B 0,C 180,E1 -1760.05,E2 -1760.05} C_VEL
LIN {X 0,Y 580.113,Z 761.724,A -85,B 0,C 180,E1 -1761.397,E2 -1761.397} C_VEL
LIN {X 0,Y 580.122,Z 755.518,A -85,B 0,C 180,E1 -1762.527,E2 -1762.527} C_VEL
LIN {X 0,Y 580.217,Z 748.179,A -85,B 0,C 180,E1 -1763.592,E2 -1763.592} C_VEL
LIN {X 0,Y 580.272,Z 738.957,A -85,B 0,C 180,E1 -1764.667,E2 -1764.667} C_VEL
LIN {X 0,Y 580.35,Z 729.114,A -85,B 0,C 180,E1 -1765.581,E2 -1765.581} C_VEL
LIN {X 0,Y 580.469,Z 718.636,A -85,B 0,C 180,E1 -1766.369,E2 -1766.369} C_VEL
LIN {X 0,Y 580.546,Z 708.388,A -85,B 0,C 180,E1 -1766.991,E2 -1766.991} C_VEL
LIN {X 0,Y 580.66,Z 696.458,A -85,B 0,C 180,E1 -1767.565,E2 -1767.565} C_VEL
LIN {X 0,Y 580.729,Z 682.727,A -85,B 0,C 180,E1 -1768.043,E2 -1768.043} C_VEL
LIN {X 0,Y 580.783,Z 670.365,A -85,B 0,C 180,E1 -1768.327,E2 -1768.327} C_VEL
LIN {X 0,Y 580.895,Z 568.59,A -85,B 0,C 180,E1 -1769.611,E2 -1769.611} C_VEL
LIN {X 0,Y 580.223,Z 564.561,A -85,B 0,C 180,E1 -1769.697,E2 -1769.697} C_VEL
LIN {X 0,Y 580.295,Z 558.2,A -85,B 0,C 180,E1 -1771.073,E2 -1771.073} C_VEL
LIN {X 0,Y 580.32,Z 558.193,A -85,B 0,C 180,E1 -1773.658,E2 -1773.658} C_VEL
LIN {X 0,Y 580.273,Z 558.207,A -85,B 0,C 180,E1 -1776.442,E2 -1776.442} C_VEL
LIN {X 0,Y 580.275,Z 558.198,A -85,B 0,C 180,E1 -1779.437,E2 -1779.437} C_VEL
LIN {X 0,Y 580.276,Z 558.198,A -85,B 0,C 180,E1 -1781.645,E2 -1781.645} C_VEL
LIN {X 0,Y 580.274,Z 558.199,A -85,B 0,C 180,E1 -1783.825,E2 -1783.825} C_VEL
LIN {X 0,Y 580.273,Z 558.206,A -85,B 0,C 180,E1 -1786.696,E2 -1786.696} C_VEL
LIN {X 0,Y 580.298,Z 558.195,A -85,B 0,C 180,E1 -1789.533,E2 -1789.533} C_VEL
LIN {X 0,Y 580.332,Z 558.198,A -85,B 0,C 180,E1 -1792.345,E2 -1792.345} C_VEL
LIN {X 0,Y 580.338,Z 558.191,A -85,B 0,C 180,E1 -1795.137,E2 -1795.137} C_VEL
LIN {X 0,Y 580.328,Z 558.192,A -85,B 0,C 180,E1 -1797.918,E2 -1797.918} C_VEL
LIN {X 0,Y 580.358,Z 558.195,A -85,B 0,C 180,E1 -1800.694,E2 -1800.694} C_VEL
LIN {X 0,Y 580.28,Z 558.196,A -85,B 0,C 180,E1 -1803.472,E2 -1803.472} C_VEL
LIN {X 0,Y 580.322,Z 558.192,A -85,B 0,C 180,E1 -1805.56,E2 -1805.56} C_VEL
LIN {X 0,Y 580.328,Z 558.198,A -85,B 0,C 180,E1 -1808.356,E2 -1808.356} C_VEL
LIN {X 0,Y 580.322,Z 558.192,A -85,B 0,C 180,E1 -1811.209,E2 -1811.209} C_VEL
LIN {X 0,Y 580.316,Z 558.194,A -85,B 0,C 180,E1 -1814.017,E2 -1814.017} C_VEL
LIN {X 0,Y 580.304,Z 558.197,A -85,B 0,C 180,E1 -1816.915,E2 -1816.915} C_VEL
LIN {X 0,Y 580.301,Z 558.195,A -85,B 0,C 180,E1 -1819.823,E2 -1819.823} C_VEL
LIN {X 0,Y 580.32,Z 558.197,A -85,B 0,C 180,E1 -1822.801,E2 -1822.801} C_VEL
LIN {X 0,Y 580.301,Z 558.196,A -85,B 0,C 180,E1 -1825.08,E2 -1825.08} C_VEL
LIN {X 0,Y 580.313,Z 558.193,A -85,B 0,C 180,E1 -1827.864,E2 -1827.864} C_VEL
LIN {X 0,Y 580.292,Z 558.202,A -85,B 0,C 180,E1 -1830.698,E2 -1830.698} C_VEL
LIN {X 0,Y 580.298,Z 558.194,A -85,B 0,C 180,E1 -1833.318,E2 -1833.318} C_VEL
LIN {X 0,Y 580.319,Z 558.193,A -85,B 0,C 180,E1 -1835.768,E2 -1835.768} C_VEL
LIN {X 0,Y 580.285,Z 558.201,A -85,B 0,C 180,E1 -1838.147,E2 -1838.147} C_VEL
LIN {X 0,Y 580.3,Z 558.199,A -85,B 0,C 180,E1 -1840.844,E2 -1840.844} C_VEL
LIN {X 0,Y 580.286,Z 558.196,A -85,B 0,C 180,E1 -1843.657,E2 -1843.657} C_VEL
LIN {X 0,Y 580.272,Z 558.207,A -85,B 0,C 180,E1 -1846.61,E2 -1846.61} C_VEL
LIN {X 0,Y 580.296,Z 558.196,A -85,B 0,C 180,E1 -1849.158,E2 -1849.158} C_VEL
LIN {X 0,Y 580.286,Z 558.198,A -85,B 0,C 180,E1 -1851.928,E2 -1851.928} C_VEL
LIN {X 0,Y 580.28,Z 558.207,A -85,B 0,C 180,E1 -1854.456,E2 -1854.456} C_VEL
LIN {X 0,Y 580.291,Z 558.199,A -85,B 0,C 180,E1 -1856.976,E2 -1856.976} C_VEL
LIN {X 0,Y 580.293,Z 558.196,A -85,B 0,C 180,E1 -1859.426,E2 -1859.426} C_VEL
LIN {X 0,Y 580.298,Z 558.201,A -85,B 0,C 180,E1 -1862.142,E2 -1862.142} C_VEL
LIN {X 0,Y 580.337,Z 558.359,A -85,B 0,C 180,E1 -1864.731,E2 -1864.731} C_VEL
LIN {X 0,Y 581.261,Z 563.41,A -85,B 0,C 180,E1 -1865.43,E2 -1865.43} C_VEL
LIN {X 0,Y 581.086,Z 583.351,A -85,B 0,C 180,E1 -1867.98,E2 -1867.98} C_VEL
LIN {X 0,Y 580.82,Z 605.034,A -85,B 0,C 180,E1 -1870.702,E2 -1870.702} C_VEL
LIN {X 0,Y 580.633,Z 627.455,A -85,B 0,C 180,E1 -1873.475,E2 -1873.475} C_VEL
LIN {X 0,Y 580.45,Z 650.794,A -85,B 0,C 180,E1 -1876.321,E2 -1876.321} C_VEL
LIN {X 0,Y 580.957,Z 655.747,A -85,B 0,C 180,E1 -1876.4,E2 -1876.4} C_VEL
LIN {X 0,Y 580.82,Z 759.962,A -85,B 0,C 180,E1 -1877.709,E2 -1877.709} C_VEL
LIN {X 0,Y 580.749,Z 772.464,A -85,B 0,C 180,E1 -1877.995,E2 -1877.995} C_VEL
LIN {X 0,Y 580.645,Z 784.919,A -85,B 0,C 180,E1 -1878.418,E2 -1878.418} C_VEL
LIN {X 0,Y 580.57,Z 795.934,A -85,B 0,C 180,E1 -1878.921,E2 -1878.921} C_VEL
LIN {X 0,Y 580.487,Z 806.588,A -85,B 0,C 180,E1 -1879.537,E2 -1879.537} C_VEL
LIN {X 0,Y 580.371,Z 817.477,A -85,B 0,C 180,E1 -1880.328,E2 -1880.328} C_VEL
LIN {X 0,Y 580.271,Z 828.115,A -85,B 0,C 180,E1 -1881.292,E2 -1881.292} C_VEL
LIN {X 0,Y 580.221,Z 835.962,A -85,B 0,C 180,E1 -1882.168,E2 -1882.168} C_VEL
LIN {X 0,Y 580.153,Z 843.651,A -85,B 0,C 180,E1 -1883.222,E2 -1883.222} C_VEL
LIN {X 0,Y 580.139,Z 850.681,A -85,B 0,C 180,E1 -1884.439,E2 -1884.439} C_VEL
LIN {X 0,Y 580.108,Z 855.372,A -85,B 0,C 180,E1 -1885.484,E2 -1885.484} C_VEL
LIN {X 0,Y 580.123,Z 858.958,A -85,B 0,C 180,E1 -1886.527,E2 -1886.527} C_VEL
LIN {X 0,Y 580.043,Z 860.81,A -85,B 0,C 180,E1 -1887.222,E2 -1887.222} C_VEL
LIN {X 0,Y 580.038,Z 862.201,A -85,B 0,C 180,E1 -1887.917,E2 -1887.917} C_VEL
LIN {X 0,Y 580.04,Z 863.785,A -85,B 0,C 180,E1 -1889.306,E2 -1889.306} C_VEL
LIN {X 0,Y 580.037,Z 864,A -85,B 0,C 180,E1 -1890,E2 -1890} C_VEL
LIN {X 0,Y 580.047,Z 863.185,A -85,B 0,C 180,E1 -1891.389,E2 -1891.389} C_VEL
LIN {X 0,Y 580.038,Z 862.2,A -85,B 0,C 180,E1 -1892.083,E2 -1892.083} C_VEL
LIN {X 0,Y 580.043,Z 860.809,A -85,B 0,C 180,E1 -1892.778,E2 -1892.778} C_VEL
LIN {X 0,Y 580.11,Z 857.896,A -85,B 0,C 180,E1 -1893.82,E2 -1893.82} C_VEL
LIN {X 0,Y 580.054,Z 853.95,A -85,B 0,C 180,E1 -1894.865,E2 -1894.865} C_VEL
LIN {X 0,Y 580.139,Z 847.878,A -85,B 0,C 180,E1 -1896.085,E2 -1896.085} C_VEL
LIN {X 0,Y 580.184,Z 841.238,A -85,B 0,C 180,E1 -1897.132,E2 -1897.132} C_VEL
LIN {X 0,Y 580.25,Z 832.992,A -85,B 0,C 180,E1 -1898.182,E2 -1898.182} C_VEL
LIN {X 0,Y 580.308,Z 824.54,A -85,B 0,C 180,E1 -1899.058,E2 -1899.058} C_VEL
LIN {X 0,Y 580.417,Z 814.099,A -85,B 0,C 180,E1 -1899.936,E2 -1899.936} C_VEL
LIN {X 0,Y 580.512,Z 803.761,A -85,B 0,C 180,E1 -1900.639,E2 -1900.639} C_VEL
LIN {X 0,Y 580.597,Z 792.241,A -85,B 0,C 180,E1 -1901.264,E2 -1901.264} C_VEL
LIN {X 0,Y 580.707,Z 779.484,A -85,B 0,C 180,E1 -1901.784,E2 -1901.784} C_VEL
LIN {X 0,Y 580.739,Z 766.451,A -85,B 0,C 180,E1 -1902.16,E2 -1902.16} C_VEL
LIN {X 0,Y 580.83,Z 754.107,A -85,B 0,C 180,E1 -1902.38,E2 -1902.38} C_VEL
LIN {X 0,Y 580.816,Z 652.17,A -85,B 0,C 180,E1 -1903.648,E2 -1903.648} C_VEL
LIN {X 0,Y 580.535,Z 649.727,A -85,B 0,C 180,E1 -1903.699,E2 -1903.699} C_VEL
LIN {X 0,Y 580.731,Z 621.487,A -85,B 0,C 180,E1 -1906.703,E2 -1906.703} C_VEL
LIN {X 0,Y 581.013,Z 594.197,A -85,B 0,C 180,E1 -1909.647,E2 -1909.647} C_VEL
LIN {X 0,Y 581.272,Z 567.537,A -85,B 0,C 180,E1 -1912.574,E2 -1912.574} C_VEL
LIN {X 0,Y 581.136,Z 561.944,A -85,B 0,C 180,E1 -1913.203,E2 -1913.203} C_VEL
LIN {X 0,Y 580.316,Z 558.202,A -85,B 0,C 180,E1 -1913.674,E2 -1913.674} C_VEL
LIN {X 0,Y 580.308,Z 558.195,A -85,B 0,C 180,E1 -1916.621,E2 -1916.621} C_VEL
LIN {X 0,Y 580.303,Z 558.196,A -85,B 0,C 180,E1 -1919.309,E2 -1919.309} C_VEL
LIN {X 0,Y 580.3,Z 558.201,A -85,B 0,C 180,E1 -1922.2,E2 -1922.2} C_VEL
LIN {X 0,Y 580.3,Z 558.195,A -85,B 0,C 180,E1 -1924.695,E2 -1924.695} C_VEL
LIN {X 0,Y 580.297,Z 558.195,A -85,B 0,C 180,E1 -1927.267,E2 -1927.267} C_VEL
LIN {X 0,Y 580.303,Z 558.201,A -85,B 0,C 180,E1 -1930.272,E2 -1930.272} C_VEL
LIN {X 0,Y 580.276,Z 558.199,A -85,B 0,C 180,E1 -1932.705,E2 -1932.705} C_VEL
LIN {X 0,Y 580.269,Z 558.2,A -85,B 0,C 180,E1 -1935.608,E2 -1935.608} C_VEL
LIN {X 0,Y 580.299,Z 558.197,A -85,B 0,C 180,E1 -1938.665,E2 -1938.665} C_VEL
LIN {X 0,Y 580.287,Z 558.196,A -85,B 0,C 180,E1 -1940.966,E2 -1940.966} C_VEL
LIN {X 0,Y 580.29,Z 558.197,A -85,B 0,C 180,E1 -1943.598,E2 -1943.598} C_VEL
LIN {X 0,Y 580.312,Z 558.199,A -85,B 0,C 180,E1 -1946.145,E2 -1946.145} C_VEL
LIN {X 0,Y 580.283,Z 558.201,A -85,B 0,C 180,E1 -1948.615,E2 -1948.615} C_VEL
LIN {X 0,Y 580.287,Z 558.195,A -85,B 0,C 180,E1 -1951.023,E2 -1951.023} C_VEL
LIN {X 0,Y 580.321,Z 558.192,A -85,B 0,C 180,E1 -1953.657,E2 -1953.657} C_VEL
LIN {X 0,Y 580.273,Z 558.206,A -85,B 0,C 180,E1 -1956.442,E2 -1956.442} C_VEL
LIN {X 0,Y 580.274,Z 558.197,A -85,B 0,C 180,E1 -1959.437,E2 -1959.437} C_VEL
LIN {X 0,Y 580.273,Z 558.197,A -85,B 0,C 180,E1 -1961.645,E2 -1961.645} C_VEL
LIN {X 0,Y 580.272,Z 558.197,A -85,B 0,C 180,E1 -1963.825,E2 -1963.825} C_VEL
LIN {X 0,Y 580.316,Z 558.193,A -85,B 0,C 180,E1 -1965.983,E2 -1965.983} C_VEL
LIN {X 0,Y 580.321,Z 558.197,A -85,B 0,C 180,E1 -1968.827,E2 -1968.827} C_VEL
LIN {X 0,Y 580.327,Z 558.189,A -85,B 0,C 180,E1 -1971.644,E2 -1971.644} C_VEL
LIN {X 0,Y 580.325,Z 558.198,A -85,B 0,C 180,E1 -1974.44,E2 -1974.44} C_VEL
LIN {X 0,Y 580.341,Z 558.19,A -85,B 0,C 180,E1 -1977.223,E2 -1977.223} C_VEL
LIN {X 0,Y 580.341,Z 558.189,A -85,B 0,C 180,E1 -1980,E2 -1980} C_VEL
LIN {X 0,Y 580.34,Z 558.199,A -85,B 0,C 180,E1 -1982.777,E2 -1982.777} C_VEL
LIN {X 0,Y 580.323,Z 558.189,A -85,B 0,C 180,E1 -1985.56,E2 -1985.56} C_VEL
LIN {X 0,Y 580.328,Z 558.193,A -85,B 0,C 180,E1 -1988.356,E2 -1988.356} C_VEL
LIN {X 0,Y 580.322,Z 558.195,A -85,B 0,C 180,E1 -1991.209,E2 -1991.209} C_VEL
LIN {X 0,Y 580.304,Z 558.195,A -85,B 0,C 180,E1 -1994.339,E2 -1994.339} C_VEL
LIN {X 0,Y 580.303,Z 558.204,A -85,B 0,C 180,E1 -1996.915,E2 -1996.915} C_VEL
LIN {X 0,Y 580.298,Z 558.194,A -85,B 0,C 180,E1 -1999.823,E2 -1999.823} C_VEL
LIN {X 0,Y 580.277,Z 558.202,A -85,B 0,C 180,E1 -2001.347,E2 -2001.347} C_VEL
LIN {X 0,Y 579.579,Z 558.286,A -85,B 0,C 180,E1 -2001.926,E2 -2001.926} C_VEL
LIN {X 0,Y 576.702,Z 558.65,A -85,B 0,C 180,E1 -2002.866,E2 -2002.866} C_VEL
LIN {X 0,Y 574.308,Z 558.943,A -85,B 0,C 180,E1 -2003.622,E2 -2003.622} C_VEL
LIN {X 0,Y 573.309,Z 559.064,A -85,B 0,C 180,E1 -2004.206,E2 -2004.206} C_VEL
LIN {X 0,Y 573.243,Z 559.073,A -85,B 0,C 180,E1 -2004.403,E2 -2004.403} C_VEL
LIN {X 0,Y 573.26,Z 559.08,A -85,B 0,C 180,E1 -2006.976,E2 -2006.976} C_VEL
LIN {X 0,Y 573.245,Z 559.076,A -85,B 0,C 180,E1 -2009.49,E2 -2009.49} C_VEL
LIN {X 0,Y 573.247,Z 559.073,A -85,B 0,C 180,E1 -2012.23,E2 -2012.23} C_VEL
LIN {X 0,Y 573.243,Z 559.076,A -85,B 0,C 180,E1 -2014.774,E2 -2014.774} C_VEL
LIN {X 0,Y 573.249,Z 559.083,A -85,B 0,C 180,E1 -2017.167,E2 -2017.167} C_VEL
LIN {X 0,Y 573.243,Z 559.077,A -85,B 0,C 180,E1 -2019.608,E2 -2019.608} C_VEL
LIN {X 0,Y 573.239,Z 559.071,A -85,B 0,C 180,E1 -2022.643,E2 -2022.643} C_VEL
LIN {X 0,Y 573.23,Z 559.079,A -85,B 0,C 180,E1 -2025.667,E2 -2025.667} C_VEL
